	m_commandHandler				: i_commandHandler;					// Command handler function (via defined interface)
	
	// FiFo Command Buffer											
	m_FiFo							: FB_MemRingBuffer;					// FIFO command buffer
	m_CommandBuffer					: ARRAY[1..M_COMMAND_BUFFER_SIZE] OF BYTE;
	
	// Finite State Machine
									
	m_CommandInterfaceFsmTable		: ARRAY [0..COMMAND_FSM_STATE_ARRAY_MAX, 0..COMMAND_FSM_EVENT_ARRAY_MAX, 0..COMMAND_FSM_ACTIONS_ARRAY_MAX] OF BYTE := [
	
	(* FsmState_ControlFault -------------------------------------------------------------------------- *)
	(*  Next State											Action		   		                     *)
	
		(* FsmEvent_ControlEnable *)
		Command_FsmState.FsmState_ControlFault,				Command_FsmAction.FsmAction_None,
                          
		(* FsmEvent_ControlDisable *)
		Command_FsmState.FsmState_ControlDisabled,			Command_FsmAction.FsmAction_DisableControl,
		
		(* FsmEvent_RunCommand *)
		Command_FsmState.FsmState_ControlFault,				Command_FsmAction.FsmAction_None,
	
		(* FsmEvent_CommandDone *)
		Command_FsmState.FsmState_ControlFault,				Command_FsmAction.FsmAction_None,

		(* FsmEvent_Fault *)  
		Command_FsmState.FsmState_ControlFault,				Command_FsmAction.FsmAction_None,
		
		(* FsmEvent_Reset *)  
		Command_FsmState.FsmState_ControlDisabled,			Command_FsmAction.FsmAction_Reset
	,
	
	(* FsmState_ControlDisabled ----------------------------------------------------------------------- *)
	(*  Next State											Action		    		                    *)
	
		(* FsmEvent_ControlEnable *)
		Command_FsmState.FsmState_ControlReady,				Command_FsmAction.FsmAction_EnableControl,
                          
		(* FsmEvent_ControlDisable *)
		Command_FsmState.FsmState_ControlDisabled,			Command_FsmAction.FsmAction_None,
		
		(* FsmEvent_RunCommand *)
		Command_FsmState.FsmState_ControlDisabled,			Command_FsmAction.FsmAction_None,
	
		(* FsmEvent_CommandDone *)
		Command_FsmState.FsmState_ControlFault,				Command_FsmAction.FsmAction_None,

		(* FsmEvent_Fault *)  
		Command_FsmState.FsmState_ControlFault,				Command_FsmAction.FsmAction_Fault,
		
		(* FsmEvent_Reset *)  
		Command_FsmState.FsmState_ControlDisabled,			Command_FsmAction.FsmAction_Reset
  	,

	(* FsmState_CommandRunning ------------------------------------------------------------------------ *)
	(*  Next State											Action				                        *)
	
		(* FsmEvent_ControlEnable *)
		Command_FsmState.FsmState_CommandRunning,			Command_FsmAction.FsmAction_None,
                          
		(* FsmEvent_ControlDisable *)
		Command_FsmState.FsmState_ControlDisabled,			Command_FsmAction.FsmAction_DisableControl,
		
		(* FsmEvent_RunCommand *)
		FSM_EVENT_INVALID,									Command_FsmAction.FsmAction_Fault,
	
		(* FsmEvent_CommandDone *)
		FSM_STATE_CONDITIONAL,								Command_FsmAction.FsmAction_CommandDone,

		(* FsmEvent_Fault *)  
		Command_FsmState.FsmState_ControlFault,				Command_FsmAction.FsmAction_Fault,
		
		(* FsmEvent_Reset *)  
		Command_FsmState.FsmState_ControlDisabled,			Command_FsmAction.FsmAction_Reset
  	,

	(* FsmState_ControlReady -------------------------------------------------------------------------- *)
	(*  Next State											Action		                    		    *)
	
		(* FsmEvent_ControlEnable *)
		Command_FsmState.FsmState_ControlReady,				Command_FsmAction.FsmAction_None,
                          
		(* FsmEvent_ControlDisable *)
		Command_FsmState.FsmState_ControlDisabled,			Command_FsmAction.FsmAction_DisableControl,
		
		(* FsmEvent_RunCommand *)
		Command_FsmState.FsmState_CommandRunning,			Command_FsmAction.FsmAction_RunCommand,
	
		(* FsmEvent_CommandDone *)
		FSM_EVENT_INVALID,									Command_FsmAction.FsmAction_Fault,

		(* FsmEvent_Fault *)  
		Command_FsmState.FsmState_ControlFault,				Command_FsmAction.FsmAction_Fault,
		
		(* FsmEvent_Reset *)  
		Command_FsmState.FsmState_ControlDisabled,			Command_FsmAction.FsmAction_Reset
		
	];
	
	m_CommandInterfacelFSM			: fb_FSM(		fsmId			:= ADR(m_CommandInterfacelFSM),
													stateTable		:= ADR(m_CommandInterfaceFsmTable),
													actionHandler	:= THIS^, 	// Use a self pointer in order to keep the action handler routine (ExecuteAction) in same function block <JAISON>
													numStates		:= Command_FsmState.NUM_FsmCommandInterfaceStates,
													numEvents		:= Command_FsmEvent.NUM_FsmCommandInterfaceEvents,
													initialState	:= Command_FsmState.FsmState_ControlDisabled);
											
	m_CommandFsmError				: BOOL;								// FSM error bit (TRUE = FSM Halted)
	m_CommandFsmErrorNum			: TFsmError;						// FSM error ENUM number
	m_CommandFsmCurrentState		: Command_FsmState;					// Current FSM state output
	m_CommandFsmLastState			: Command_FsmState;					// Previous state used for debugging FSM errors
	m_CommandFsmLastEvent			: Command_FsmEvent;					// Last triggered event output
	m_CommandFsmLastAction			: Command_FsmAction;				// Last run action output
	
	m_CommandFsmTraceTable			: ARRAY[1..20] OF Command_FsmDebugTableEntry;
	
END_VAR
VAR CONSTANT
	(* DEFAULT COMMAND DEFINITIONS *)
	
	(* ----------------------------------------------------------------------------
	Const name  : M_COMMAND_NONE
	Description : Defined constant value for no command running.		
	Notes       : 
	---------------------------------------------------------------------------- *)
	M_COMMAND_NONE			: INT := 0;

	(* ----------------------------------------------------------------------------
	Const name  : M_COMMAND_RESET
	Description : Defined constant value for reset command.				
	Notes       : 
	---------------------------------------------------------------------------- *)
	M_COMMAND_RESET			: INT := -1;	
	
	(* ----------------------------------------------------------------------------
	Const name  : M_COMMAND_FAULT
	Description : Defined constant value for fault command.				
	Notes       : 
	---------------------------------------------------------------------------- *)
	M_COMMAND_FAULT			: INT := -2;	

		(* ----------------------------------------------------------------------------
	Const name  : M_RESPONSE_READY
	Description : Defined constant value for ready response.		
	Notes       : 
	---------------------------------------------------------------------------- *)
	M_RESPONSE_READY		: INT := 0;

	(* ----------------------------------------------------------------------------
	Const name  : M_RESPONSE_BUSY
	Description : Defined constant value for busy response.				
	Notes       : 
	---------------------------------------------------------------------------- *)
	M_RESPONSE_BUSY			: INT := -1;	
	
	(* ----------------------------------------------------------------------------
	Const name  : M_RESPONSE_FAULT
	Description : Defined constant value for fault response.				
	Notes       : 
	---------------------------------------------------------------------------- *)
	M_RESPONSE_FAULT		: INT := -2;	
	
	
	(* FIFO COMMAND BUFFER *)
	
	(* ----------------------------------------------------------------------------
	Const name  : M_COMMAND_BUFFER_NUM_ENTRIES
	Description : Maximum number of entries allocated for the FIFO buffer.			
	Notes       : Used in FIFO buffer size definition
	---------------------------------------------------------------------------- *)
	M_COMMAND_BUFFER_NUM_ENTRIES	: UINT := 20;
		
	(* ----------------------------------------------------------------------------
	Const name  : M_COMMAND_BUFFER_SIZE
	Description : Size in BYTES allocated for the FIFO buffer.			
	Notes       : Used in FIFO buffer initialization, Beckhoff adds 4 BYTES
				  to each entry into the buffer because each data set is complemented 
				  with additional information, so that it can be located later.
	---------------------------------------------------------------------------- *)
	M_COMMAND_BUFFER_SIZE	: UINT := M_COMMAND_BUFFER_NUM_ENTRIES * (SIZEOF(TControlCommandBuffer) + 4);
	
	(* Finite State Machine *)

	(* ----------------------------------------------------------------------------
	Const name  : FSM_NUM_EVENT_ACTIONS
	Description : Maximum number of actions that are to be executed for each event 
				  Must be at least 1 action defined				
	Notes       : Used in FSM table definitions
	---------------------------------------------------------------------------- *)
	COMMAND_FSM_NUM_EVENT_ACTIONS	: INT := 1;
	
	(* ----------------------------------------------------------------------------
	Const name  : FSM_NUM_STATES
	Description : Total number of states 
	Notes       : Used in FSM table definitions
	---------------------------------------------------------------------------- *)
	COMMAND_FSM_NUM_STATES			: INT := Command_FsmState.NUM_FsmCommandInterfaceStates;
	
	(* ----------------------------------------------------------------------------
	Const name  : FSM_NUM_EVENTS
	Description : Total number of events per state
	Notes       : Used in FSM table definitions
	---------------------------------------------------------------------------- *)
	COMMAND_FSM_NUM_EVENTS			: INT := Command_FsmEvent.NUM_FsmCommandInterfaceEvents;
	
	(* ----------------------------------------------------------------------------
	Const name  : FSM_STATE_ARRAY_MAX
	Description : Max state array index value in the FSM table
				  Must subtract 1 due to arrays starting at 0
	Notes       : Used in FSM table definitions
	---------------------------------------------------------------------------- *)
	COMMAND_FSM_STATE_ARRAY_MAX		: INT := COMMAND_FSM_NUM_STATES - 1;
	
	(* ----------------------------------------------------------------------------
	Const name  : FSM_EVENT_ARRAY_MAX
	Description : Max event array index value in the FSM table
				  Must subtract 1 due to arrays starting at 0
	Notes       : Used in FSM table definitions
	---------------------------------------------------------------------------- *)
	COMMAND_FSM_EVENT_ARRAY_MAX		: INT := COMMAND_FSM_NUM_EVENTS - 1;
	
	(* ----------------------------------------------------------------------------
	Const name  : FSM_ACTIONS_ARRAY_MAX
	Description : Max actions array index value in the FSM table
				  next state entry is element 0 
	Notes       : Used in FSM table definitions
	---------------------------------------------------------------------------- *)
	COMMAND_FSM_ACTIONS_ARRAY_MAX	: INT := COMMAND_FSM_NUM_EVENT_ACTIONS;
END_VAR

(* ---------------------------------------------------------------------------
Func name   : 	CMD_ClearCommandBuffer
Description : 	Resets the FIFO buffer and clears current command and
				all buffered commands.
Inputs      :	None
Returns     : 	TRUE
Notes       : 	Used when the command interface is reset.
--------------------------------------------------------------------------- *)

METHOD CMD_ClearCommandBuffer : BOOL
VAR_INPUT
END_VAR
// Clear the command buffer			
MEMSET			(	destAddr:= ADR(m_CommandBuffer) , 
				 	fillByte:= 0 , 
				 	n:= SIZEOF(m_CommandBuffer));	

// Clear the current command variable		
MEMSET			(	destAddr:= ADR(m_CurrentCommand) , 
				 	fillByte:= 0 , 
					n:=  SIZEOF(m_CurrentCommand));	

// Reset the command buffer					
m_FiFo.A_Reset();

CMD_ClearCommandBuffer := TRUE;
END_METHOD

(* ---------------------------------------------------------------------------
Func name   : 	CMD_Fault
Description : 	Faults the FSM and transitions to the "Fault" state.
				Commands will NO LONGER be processed.
Inputs      :	None
Returns     : 	None
Notes       : 	Can be used in the interface routines if an error
				occurs that warrants command processing to stop.
--------------------------------------------------------------------------- *)

METHOD CMD_Fault
VAR_INPUT
END_VAR
// FAULT- Send Fault event to FSM
m_CommandInterfacelFSM.FSM_ProcessEvent(event:= Command_FsmEvent.FsmEvent_Fault);
END_METHOD

(* ---------------------------------------------------------------------------
Func name   : 	CMD_Init
Description : 	Initialization routine to setup the command interface
Inputs      :	commandHandler	:	command handler functions pointer (via defined interface)
Returns     : 	None
Notes       : 	Should be run ONCE for each instantiation of the
				command interface. Usually in the FB_INIT method.
--------------------------------------------------------------------------- *)

METHOD CMD_Init
VAR_INPUT
	commandHandler		: i_commandHandler;		// Command handler function (via defined interface)
END_VAR
// Set the FSM error state
m_CommandInterfacelFSM.FSM_SetErrorState(Command_FsmState.FsmState_ControlFault);

// Clear all event triggers to ensure all events are captured on startup
m_EnableTrigger(CLK:= FALSE);
m_DisableTrigger(CLK:= FALSE);
m_CommandDoneTrigger(CLK:= FALSE);

// Clear all flags
xBusy 	:= FALSE;
xDone 	:= FALSE;
xFault	:= FALSE;

// Set initial Variables
m_ControlEnabled := FALSE;

// Initialize the Command Handler Function
m_commandHandler := commandHandler;

// FIFO initialization - Not Needed <REMOVE>
//m_FiFo.Initialize(pBuffer := ADR(m_CommandBuffer[1]), udiBufferSize := M_COMMAND_BUFFER_SIZE * SIZEOF(TControlCommandBuffer));
//m_FiFo(pBuffer := ADR(m_CommandBuffer[1]), cbBuffer := M_COMMAND_BUFFER_SIZE * SIZEOF(TControlCommandBuffer)); // TEST THIS

// Fsm Test Table
m_CommandInterfacelFSM.FSM_SetDebugTraceTable(	pDebugTable := ADR(m_CommandFsmTraceTable),
												uiTableSize := SIZEOF(m_CommandFsmTraceTable));
END_METHOD

(* ---------------------------------------------------------------------------
Func name   : 	CMD_IsCommandValid
Description : 	Determines the validity of a command input.
Inputs      :	command	:	command to check of type TControlCommand (INT)
Returns     : 	TRUE if command is valid, FALSE otherwise
Notes       : 	Valid commands are > 0
--------------------------------------------------------------------------- *)

METHOD CMD_IsCommandValid : BOOL
VAR_INPUT
	command		: TControlCommand;
END_VAR
// Check for valid command which is greater than 0.  
// NONE (0) and RESET (-1) are handled seperately. <JAISON>
IF command > 0 THEN
			
	CMD_IsCommandValid := TRUE;
				
ELSE
		
	// COMMAND INVALID
	CMD_IsCommandValid := FALSE;
		
END_IF
END_METHOD

(* ---------------------------------------------------------------------------
Func name   : 	CMD_Reset
Description : 	Sends reset command to the FSM and clears the trace table
				if configured.
Inputs      :	None
Returns     : 	None
Notes       : 	
--------------------------------------------------------------------------- *)

METHOD CMD_Reset
VAR_INPUT
END_VAR
// Send the Reset Command event to FSM
m_CommandInterfacelFSM.FSM_ProcessEvent(event:= Command_FsmEvent.FsmEvent_Reset);

// Clear the trace table
IF (m_pCmdTraceTable <> _NULL) THEN					
	MEMSET			(	destAddr	:= ADR(m_pCmdTraceTable) , 
						fillByte	:= 0 , 
				 		n			:=  SIZEOF(m_CmdTraceTableSize));	
END_IF
END_METHOD

(* ---------------------------------------------------------------------------
Func name   : 	CMD_SendCommand
Description : 	Sends the input command with Parms to the FIFO buffer
				to be processed by the interface.
Inputs      :	command	:	command ENUM type TControlCommand (INT)
				parms	:	pointer to command PARMS of type TControlCommandParms (ARRAY[1..12] OF WORD)
Returns     : 	TRUE on success, FALSE otherwise
Notes       : 	
--------------------------------------------------------------------------- *)

METHOD CMD_SendCommand : BOOL
VAR_INPUT
	command		: TControlCommand;
	parms		: POINTER TO TControlCommandParms;
END_VAR
VAR
	m_Command	: TControlCommandBuffer;
END_VAR
VAR CONSTANT
	nullParms	: TControlCommandParms := [0, 0, 0, 0, 0, 0, 0, 0, 0, 0, 0, 0];
END_VAR
// Handle special case of Reset Command - sends command directly to FSM
IF (command = M_COMMAND_RESET) THEN
	
	// Send the Reset Command event to FSM
	m_CommandInterfacelFSM.FSM_ProcessEvent(event:= Command_FsmEvent.FsmEvent_Reset);
	
	CMD_SendCommand := TRUE;

// Handle special case of None Command
ELSIF (command = M_COMMAND_NONE) THEN
	
	// DO NOTHING
	
	CMD_SendCommand := TRUE;
	
ELSIF (command = M_COMMAND_FAULT) THEN
	
	CMD_Fault();
	
	CMD_SendCommand := TRUE;

ELSIF (m_FiFo.nCount < M_COMMAND_BUFFER_NUM_ENTRIES) AND m_ControlEnabled AND CMD_IsCommandValid(command) THEN

	m_Command.command := command;
	
	IF (parms <> _NULL) THEN
		m_Command.parms := parms^;
	ELSE
		m_Command.parms := nullParms;
	END_IF
	
	// Clear Response Here
	MEMSET			(	destAddr	:= ADR(m_Command.response), 
						fillByte	:= 0, 
						n			:= SIZEOF(m_Command.response));
								
	m_FiFo.A_AddTail(pWrite := ADR(m_Command), cbWrite := SIZEOF(m_Command));
	
	CMD_SendCommand := TRUE;

ELSE
	
	CMD_SendCommand := FALSE;
	
END_IF
END_METHOD

(* ---------------------------------------------------------------------------
Func name   : 	CMD_SetTraceTable
Description : 	Sets the trace table for use with the CMD_TRACE function which
				tracks previously completed commands.
Inputs      :	pTraceTable			-	pointer to the trace table
				uiTableSize			-	size of the trace table array in BYTES
Returns     : 	TRUE on success, else FALSE
Notes       : 	When setting a trace table use the generic TControlCommandBuffer
				type in order to ensure the size is proper.  The derived class
				will be responsible for decoding the command/response INT values
				into more understandable ENUMs if required.
--------------------------------------------------------------------------- *)

METHOD CMD_SetTraceTable : BOOL
VAR_INPUT
	pTraceTable			: POINTER TO TControlCommandBuffer;		// Pointer to the trace table
	uiTableSize			: UINT;									// Size of the debug table array in BYTES
END_VAR
// Test to ensure the debug table size is dividible by BYTES so the pointer manipulation does not crash the system. <JAISON>
IF ((uiTableSize MOD SIZEOF(TControlCommandBuffer)) = 0) THEN
	
	// Clear the trace table				
	MEMSET		     (	destAddr	:= 	pTraceTable, 
				 		fillByte	:= 0 , 
						n			:=  uiTableSize);	

	// Set the trace table pointer
	m_pCmdTraceTable := pTraceTable;
	
	// Set the trace table size
	m_CmdTraceTableSize := uiTableSize;
	
	// Return TRUE
	CMD_SetTraceTable := TRUE;
	
ELSE
	
	// Return FALSE
	CMD_SetTraceTable := FALSE;
	
END_IF
END_METHOD

(* ---------------------------------------------------------------------------
Func name   : 	CMD_TRACE
Description : 	This method allows the command interface to trace previously
				completed commands in an externally defined trace table.
Inputs      :	command	-	pointer to the command buffer to be added
Returns     : 	None
Notes       : 	Initially the trace table pointer will be NULL, you must 
				run the CMD_SetTraceTable to initialize the functionality.
--------------------------------------------------------------------------- *)
METHOD CMD_TRACE

VAR_INPUT
	command 			: POINTER TO TControlCommandBuffer;	// The command to be added to the trace table
END_VAR
VAR
	m_NumCommands		: UINT;								// Calculated number of commands in the trace table
	m_Command			: TControlCommandBuffer;			// Copy of the current command
	Offset				: UINT;								// Trace table pointer offset variable
	pCurrent 			: POINTER TO TControlCommandBuffer;	// Pointer to the current array element, used for array shifting
	pPrevious			: POINTER TO TControlCommandBuffer;	// Pointer to the previous array element, used for array shifting
END_VAR
// Ensure the trace table has been initialized
IF ((m_pCmdTraceTable <> _NULL) AND (command <> _NULL)) THEN
	
	// Determine the number of commands in the debug table array
	m_NumCommands := m_CmdTraceTableSize / SIZEOF(TControlCommandBuffer);
	
	// Set the offset to point to the last element of the debug table array
	Offset := (m_NumCommands - 1) * SIZEOF(TControlCommandBuffer);
	
	// Shift all the previous states down by one element
	WHILE (Offset >  0) DO
		
		// Set the current and previous state pointers
		pCurrent := m_pCmdTraceTable + Offset;
		pPrevious := pCurrent - SIZEOF(TControlCommandBuffer);
		
		// Update the current state value to the previous value
		pCurrent^ := pPrevious^;
	
		// Move the offset up by one element
		Offset := Offset - SIZEOF(TControlCommandBuffer);
		
	END_WHILE
	
	// Copy command data to local variable					
	MEMCPY		( destAddr := ADR(m_Command),
				  srcAddr  := command,
				  n		   := SIZEOF(m_Command));	
				  
	// Set the current state as the first element in the debug trace table array
	m_pCmdTraceTable^ := m_Command;
	
END_IF
END_METHOD

(* ---------------------------------------------------------------------------
Func name   : 	CMD_UpdateCommandInterface
Description : 	Interface update routine which is required to be called
				on EACH PLC SCAN by the inherited class.  This method is
				responsible for updating the FIFO buffer and FSM.
Inputs      :	None
Returns     : 	None
Notes       : 	
--------------------------------------------------------------------------- *)

METHOD CMD_UpdateCommandInterface
VAR_INPUT
END_VAR
//Run the Module Finite State Machine Logic Block <JAISON>
m_CommandInterfacelFSM(xEnable:= xEnable, xError=> m_CommandFsmError, errorNum=> m_CommandFsmErrorNum);

//Set the current FSM State variable for testing the FSM state transitions <JAISON>
m_CommandFsmCurrentState := m_CommandInterfacelFSM.FSM_GetCurrentState();

m_CommandFsmLastState := m_CommandInterfacelFSM.FSM_GetPreviousState();

// Run the Module FiFo Buffer Logic Block <JAISON>
m_FiFo(	pBuffer		:= ADR(m_CommandBuffer), 
		cbBuffer	:= M_COMMAND_BUFFER_SIZE);

// Handle the FIFO command buffer ONLY when in the ModuleReady state
IF (m_FiFo.nCount > 0) AND (m_CommandFsmCurrentState = Command_FsmState.FsmState_ControlReady) THEN
	
	// Remove an element from the command buffer <JAISON>
	m_FiFo.A_RemoveHead(pRead:= ADR(m_CurrentCommand), cbRead:= SIZEOF(m_CurrentCommand));
	
	// Ensure command is valid
	// This step is superfluous as commands going into the buffer are screened,
	// however, this should catch any data issues with the buffer. <JAISON>
	IF CMD_IsCommandValid(m_CurrentCommand.command) THEN
		
		// Send the Run Command event to FSM - Parm is pointer to the current command
		m_CommandInterfacelFSM.FSM_ProcessEventWithParms(	event		:= Command_FsmEvent.FsmEvent_RunCommand, 
															parms		:= ADR(m_CurrentCommand), 
															parmSize	:= SIZEOF(ADR(m_CurrentCommand)));
	
	ELSE
		
		// Send Fault event to FSM
		m_CommandInterfacelFSM.FSM_ProcessEvent(event:= Command_FsmEvent.FsmEvent_Fault);
		
	END_IF
	
END_IF

// (* EVENT TRIGGERS *)

// Module enable trigger, basic FSM Event with no user parameters <JAISON>
m_EnableTrigger(CLK:= xEnable);
IF (m_EnableTrigger.Q)THEN
	m_CommandInterfacelFSM.FSM_ProcessEvent(event:= Command_FsmEvent.FsmEvent_ControlEnable);
END_IF

// Module disable trigger, basic FSM Event with no user parameters <JAISON>
m_DisableTrigger(CLK:= xEnable);
IF (m_DisableTrigger.Q)THEN
	m_CommandInterfacelFSM.FSM_ProcessEvent(event:= Command_FsmEvent.FsmEvent_ControlDisable);
END_IF

// Handle command continuous logic HERE
IF (xBusy) THEN
	m_CommandDoneTrigger(CLK:= m_commandHandler.CommandRunning(pCurrentCommand:= ADR(m_CurrentCommand)));
ELSE
	m_CommandDoneTrigger(CLK:= FALSE);
END_IF

// Command done trigger, basic FSM Event with no user parameters <JAISON>
IF (m_CommandDoneTrigger.Q)THEN
	m_CommandInterfacelFSM.FSM_ProcessEventWithParms(	event		:= Command_FsmEvent.FsmEvent_CommandDone, 
														parms		:= ADR(m_CurrentCommand), 
														parmSize	:= SIZEOF(ADR(m_CurrentCommand)));
END_IF
END_METHOD

(* ---------------------------------------------------------------------------
Func name   : 	ExecuteAction
Description : 	This method is a standardized handler for
				each action generated by the FSM
Inputs      :	p_FSM			-	pointer to the instantiation of the FSM object
				currentAction	-	current FSM action being processed
				currentEvent	-	current FSM event being processed
Returns     : 	BOOL			- 	result of action function
Notes       : 	The approach of using an interface enables the user 
				of the FSM to define and handle actions based 
				on their design and implementation.
				
				Return TRUE to change state, FALSE to remain in 
				the same state, unless the FSM has the alwaysChangeState
				set to TRUE, then it will change state regardless 
				of action handler return.
				
				If a conditional state is to be used this action handler
				routuine is responsible for setting the conditionalState 
				value using the FSM_SetConditionalState() function.
--------------------------------------------------------------------------- *)

METHOD ExecuteAction : BOOL
VAR_INPUT
	p_FSM			: POINTER TO fb_FSM;
	currentAction	: TFsmAction;
	currentEvent	: TFsmEventDesc;
END_VAR
VAR
	pCurrentCommand	: POINTER TO TControlCommandBuffer;		// Pointer to current command parms
	faultCommand	: TControlCommandBuffer;				// Fault command buffer
	resetCommand	: TControlCommandBuffer;				// Reset command buffer
END_VAR
CASE currentAction OF
		
	Command_FsmAction.FsmAction_None:
			
		// DO ACTION NONE
			
		// RETURN TRUE
		ExecuteAction := TRUE;
			
	Command_FsmAction.FsmAction_EnableControl:
		
		// DO ACTION ENABLE CONTROL
				
		CMD_ClearCommandBuffer();
		xDone 	:= FALSE;
		xBusy	:= FALSE;
		xFault	:= FALSE;
			
		// Enable the control
		m_ControlEnabled := TRUE;
			
		// RETURN TRUE
		ExecuteAction := TRUE;
		
	Command_FsmAction.FsmAction_DisableControl:
		
		// DO ACTION DISABLE CONTROL
			
		CMD_ClearCommandBuffer();
		xDone := FALSE;
		xBusy := FALSE;
			
		// Disable the control
		m_ControlEnabled := FALSE;
			
		// RETURN TRUE
		ExecuteAction := TRUE;
			
	Command_FsmAction.FsmAction_RunCommand:
		
		// DO ACTION RUN COMMAND
			
		// Event Parms are pointer to TControlCommandBuffer
		pCurrentCommand := currentEvent.parms;
			
		// Clear the last run command response
		MEMSET(				destAddr	:= ADR(pCurrentCommand^.response), 
							fillByte	:= 0 , 
							n			:=  SIZEOF(pCurrentCommand^.response));	
				
		// Set the response to show command is running
		pCurrentCommand^.response.response 	:= M_RESPONSE_BUSY;
		pCurrentCommand^.response.message 	:= TO_STRING("Command Running");
		
		// Handle command start logic HERE 
		IF (NOT m_commandHandler.CommandStart(pCurrentCommand:= pCurrentCommand)) THEN
									
			// COMMAND START ERROR - Send Fault event to FSM
			m_CommandInterfacelFSM.FSM_ProcessEvent(event:= Command_FsmEvent.FsmEvent_Fault);
			
		END_IF
			
		// Set output flags
		xBusy := TRUE;
		xDone := FALSE;
			
		// Reset command done flag
		m_CommandDoneTrigger(CLK:= FALSE);
			
		// RETURN TRUE
		ExecuteAction := TRUE;
			
	Command_FsmAction.FsmAction_CommandDone:
		
		// DO ACTION COMMAND DONE - CONDITIONAL STATE
			
		// Event Parms are pointer to TControlCommandBuffer
		pCurrentCommand := currentEvent.parms;
		
		// Handle command done logic HERE - Set the response - Set the next state
		IF (m_commandHandler.CommandDone(pCurrentCommand:= pCurrentCommand)) THEN
				
			p_FSM^.FSM_SetConditionalState(state:= Command_FsmState.FsmState_ControlReady);
			
		ELSE
			
			// COMMAND DONE ERROR - Send Fault event to FSM
			m_CommandInterfacelFSM.FSM_ProcessEvent(event:= Command_FsmEvent.FsmEvent_Fault);
			
		END_IF
			
		// Set output flags
		xBusy := FALSE;
		xDone := TRUE;
			
		// Reset command done flag
		m_CommandDoneTrigger(CLK:= FALSE);
						
		// Add the current command/response to the trace table
		CMD_TRACE(command:= pCurrentCommand);
			
		// RETURN TRUE
		ExecuteAction := TRUE;
			
	Command_FsmAction.FsmAction_Fault:
		
		// DO ACTION FAULT
			
		// Disable the control
		m_ControlEnabled := FALSE;
		
		xFault	:= TRUE;
			
		// Modify the current response message to show fault
		m_CurrentCommand.response.response	:= M_RESPONSE_FAULT;
		m_CurrentCommand.response.message	:= TO_STRING("COMMAND INTERFACE FAULTED");
			
		// Copy the current command data, to show the command 
		// running when the fault occured; if any.		
		faultCommand.command 			:= m_CurrentCommand.command;
		faultCommand.parms				:= m_CurrentCommand.parms;
	
		// Modify the response to show that this is a fault event
		faultCommand.response.response 	:= M_RESPONSE_FAULT;
		faultCommand.response.message 	:= TO_STRING("COMMAND INTERFACE FAULTED");
			
		CMD_TRACE(command:= ADR(faultCommand));
			
		// Call Interface Fault function
		m_commandHandler.Fault();
			
		// RETURN TRUE
		ExecuteAction := TRUE;
		
	Command_FsmAction.FsmAction_Reset:
		
		// DO ACTION RESET
			
		CMD_ClearCommandBuffer();
			
		xDone 	:= FALSE;
		xBusy 	:= FALSE;
		xFault	:= FALSE;
			
		// Copy the current command data, to show the command 
		// is a reset command		
		resetCommand.command 			:= M_COMMAND_RESET;
	
		// Modify the response to show that the reset occured
		resetCommand.response.response 	:= M_RESPONSE_READY;
		resetCommand.response.message 	:= TO_STRING("COMMAND INTERFACE RESET");
			
		CMD_TRACE(command:= ADR(resetCommand));
		
		// Call Interface Reset function
		m_commandHandler.Reset();
			
		// Reset enable trigger to capture enable event
		m_EnableTrigger(CLK:= FALSE);
			
		// RETURN TRUE
		ExecuteAction := TRUE;	
				
	FSM_ACTION_UNEXPECTED_EVENT:
			
		// DO ACTION UNEXPECTED EVENT
		
		// ERROR TRAP - UNKNOWN ACTION
		// NOTE: 	This will HALT the FSM when it FAILS which is likely advisable here because
		//			this is a critical design time error.  All actions need to be defined, even
		//			if they simply log an event occured. <JAISON>
		p_FSM^.FSM_ASSERT(FALSE, TFsmError.FSM_INVALID_ACTION);
			
		// RETURN FALSE
		ExecuteAction := FALSE;
			
	FSM_ACTION_ERROR_EVENT:
		
		// DO ACTION ERROR EVENT
			
		// This action is executed when an FSM ASSERT Fails and the FSM is transitioning to the defined error state. <JAISON>
			
		// RETURN FALSE - This is irrelevant because the FSM will automatically transition to the error state.
		ExecuteAction := FALSE;
				
ELSE
			
	// ERROR TRAP - UNKNOWN ACTION
	// NOTE: 	This will HALT the FSM when it FAILS which is likely advisable here because
	//			this is a critical design time error.  All actions need to be defined, even
	//			if they simply log an event occured. <JAISON>
	p_FSM^.FSM_ASSERT(FALSE, TFsmError.FSM_INVALID_ACTION);
			
	// RETURN FALSE
	ExecuteAction := FALSE;
			
END_CASE;
	
m_CommandFsmLastEvent := currentEvent.event;
m_CommandFsmLastAction := currentAction;
m_CommandFsmLastState := p_FSM^.FSM_GetPreviousState();
END_METHOD

END_FUNCTION_BLOCK

// 20 Program Organization Units/FSM/Interfaces/i_actionHandler
(*AUTHOR:			Jaison Schaab*)
(*DATE:				December. 30 / 2019*)
(*DESCRIPTION: 		This is a standardized interface used by the FSM function
					block to handle generated actions*)
					
(*NOTES:      	 	All methods definied by this interface are required to
					be implimented by the user defined action handler
					function block.  Each methods inputs/outputs need
					to match exactly what is defined by the interface.
					
					The FSM requires the user defined function block which
					impliments this interface  to be passed into its 
					constructor upon instantiation.*)

INTERFACE i_actionHandler

(* ---------------------------------------------------------------------------
Func name   : 	ExecuteAction
Description : 	This method is a standardized handler for
				each action generated by the FSM
Inputs      :	p_FSM			-	pointer to the instantiation of the FSM object
				currentAction	-	current FSM action being processed
				currentEvent	-	current FSM event being processed
Returns     : 	BOOL			- 	result of action function
Notes       : 	The approach of using an interface enables the user 
				of the FSM to define and handle actions based 
				on their design and implementation.
				
				Return TRUE to change state, FALSE to remain in 
				the same state, unless the FSM has the alwaysChangeState
				set to TRUE, then it will change state regardless 
				of action handler return.
				
				If a conditional state is to be used this action handler
				routuine is responsible for setting the conditionalState 
				value using the FSM_SetConditionalState() function.
--------------------------------------------------------------------------- *)

METHOD ExecuteAction : BOOL
VAR_INPUT
	p_FSM			: POINTER TO fb_FSM;
	currentAction	: TFsmAction;
	currentEvent	: TFsmEventDesc;
END_VAR
END_METHOD

END_INTERFACE

// 20 Program Organization Units/FSM/fb_FSM
(*AUTHOR:			Jaison Schaab*)
(*DATE:				December 30 / 2019*)
(*DESCRIPTION: 		This Function Block provides a standard base functionality for
					a generic table driven finite state machine (FSM)*)
					
(*NOTES:			The user of the FSM function block is required to define the following:
					STATE ENUM of TYPE FsmState (BYTE) 		- 	List of desired states starting at 0 with the last entry being "NUM_FsmTestStates"
					EVENT ENUM of TYPE FsmEvent (BYTE) 		- 	List of desired events starting at 0 with the last entry being "NUM_FsmTestEvents"
					ACTION ENUM of TYPE FsmAction (BYTE) 	- 	List of desired actions starting at 0 with the last entry being "NUM_FsmTestActions"
					
					****The IEC Standard does NOT allow the ENUMERATION types to be defined as a non-registered type (ex. FsmState)
						To work around this simply define the required ENUMERATIONS as BYTE and remove the 
						"{attribute 'strict'}" from the header so that the system will correlate the non-registered types****
					
					Action Handler function block  			- 	user defined function block which impliments the i_actionHandler interface and
																will perform all required actions that are associated with events.
																
					****EVENTS may have parameters associated with them, ACTIONS DO NOT.  The user is required to define their own
						parameter types which can be associated with events and passed into the action handler.****									
					
					****TO TRIGGER EVENTS use the FSM methods "FSM_ProcessEvent" OR "FSM_ProcessEventWithParms"****
					****Calling the "FSM_Reset" method will RESET the FSM back to the default constructor state
						This is required after any FSM error as the FSM block will cease to function until a RESET occurs****
*)

(*UPDATE: 			March. 18 2021 - Jaison Schaab

					Code Ported from Wago.
					
					Code has NOT Yet been tested.
*)

FUNCTION_BLOCK fb_FSM
VAR_INPUT
	xEnable				: BOOL;											// Function block enable - TRUE to enable FSM functionality
END_VAR
VAR_OUTPUT
	xError				: BOOL;											// FSM error state output, if TRUE FSM will cease operation until reset (FSM_ASSERT sets state)
	errorNum			: TFsmError;									// The enumeration value describing the failed assert (type FsmError) 
END_VAR
VAR
	(* Fsm Desc *)
	m_fsmId				: POINTER TO fb_FSM;							// Pointer to the instantiation of the FSM object
	
	m_currentState		: TFsmState;									// Current state id of the FSM
	m_prevState			: TFsmState;									// Memory of the previously ran state used for debugging errors
	m_initialState		: TFsmState;									// Internal memory of the initial state id, used for FSM reset
	m_errorState		: TFsmState;									// Internal memory of an error state id, used when FSM Assert fails
	
	m_conditionalState	: TFsmState;									// Conditional next state parameter - set by action handler
	m_alwaysChangeState	: BOOL;											// Internal state change flag for conditional states - when TRUE action handler return is ignored
	
	m_numStates			: UINT;											// Number of states in the FSM
	m_numEvents			: UINT;											// Number of events defined for the FSM
	
	m_stateTable		: POINTER TO TFsmState;							// Pointer to the FSM table
	m_eventEntrySize	: UINT;											// Size of an event entry in the FSM table, consists of one event type and one action type
	m_stateEntrySize	: UINT;											// Size of a state entry in the FSM table, consists of numEvents * event entry size
	
	m_eventQ			: ARRAY[0.._FSM_EVENT_Q_SIZE] OF TFsmEventDesc;	// Event queue array, utilized as a circular buffer
	m_eventQPutIndex	: TFsmEventQIndex;								// Event queue index used for inserting events
	m_eventQGetIndex	: TFsmEventQIndex;								// Event queue index used for removing events
	m_numInEventQ		: TFsmEventQIndex;								// Current number of events in the queue
	
	m_FsmActionHandler	: i_actionHandler;								// Action handler function (via defined interface)
	
	(* Internal *)
	m_nextState 		: TFsmState;									// Internal variable used to track the next state transition
	m_changeState		: BOOL := TRUE;									// Internal state change flag used when processing events
	m_currentEvent		: TFsmEventDesc;								// Current FSM event being processed
	m_currentAction		: TFsmAction;									// Current FSM action id being processed
	
	m_pFsmDebugTable	: POINTER TO TFsmDebugTableEntry;				// Pointer to the debug table
	m_FsmDebugTableSize	: UINT;											// Size of the debug table array in BYTES
	m_StateChangeTimer	: fb_ElapsedTime;								// Timer to track the time between state changes in debug table
	
END_VAR

(* Handle the events *)
WHILE ((xEnable) AND (m_numInEventQ <> 0) AND (NOT xError)) DO
  
	m_changeState := TRUE;						// Assume we are going to change state
	m_conditionalState := FSM_STATE_INVALID; 	// Assume the conditional state is invalid to ensure the action function sets it
	
	m_currentEvent := FSM_GetCurrentEvent();
	m_currentAction := FSM_GetCurrentAction(state:= m_currentState, event:= m_currentEvent);
	
	m_prevState := m_CurrentState;				// Set the previous state for debugging FSM errors
	
	(* FSM TRACE HANDLE EVENT *)
	
	(* unexpected action, do not change state *)
	IF (m_currentAction = FSM_ACTION_UNEXPECTED_EVENT) THEN
		
		(* FSM TRACE UNEXPECTED ACTION *)
		m_changeState := FALSE;	
	
	END_IF
	
	(* FSM TRACE EXECUTE ACTION *)
	
	(* process the action, returning true means change state, but check the change state flag *)
	IF (NOT m_FsmActionHandler.ExecuteAction(p_FSM:= m_fsmId, currentAction:= m_currentAction, currentEvent:= m_currentEvent)) THEN
		
		// Action Handler Returned FALSE
		IF (_FSM_ALLOW_CONDITIONAL_STATES) THEN
			
			(* maybe change state on a FALSE return *)
			IF (m_alwaysChangeState =  FALSE) THEN
					
				m_changeState := FALSE;
				
			END_IF
				
		ELSE
			
		// Never change state on a FALSE return
        m_changeState := FALSE;
			
		END_IF
		
	END_IF (* end - (actions) *)
	
	(* Change state *)
	IF (m_changeState) THEN
    
		m_nextState := FSM_GetNextState(state:= m_currentState, event:= m_currentEvent);

		(* 	get the next state dynamically from the action handler 
			if allowed and conditional state entered into table. *)
		IF ((_FSM_ALLOW_CONDITIONAL_STATES) AND (m_nextState = FSM_STATE_CONDITIONAL)) THEN

			m_nextState := m_conditionalState;
		
		END_IF
      
		(* validate the next state value *)
		FSM_ASSERT(BYTE_TO_UINT(m_nextState) < m_numStates, TFsmError.FSM_INVALID_NEXT_STATE);
		
		// If next state is invalid, stay in same state - Assert above will set xError flag
		// Ignore this if the FSM_ASSERT already set the current state to the error state <JAISON>
		IF ((xError) AND (m_currentState <> m_errorState) )THEN
			(* stay in the same state *)
			m_nextState := m_currentState;
		END_IF
    
	ELSE
    
		(* stay in the same state *)
		m_nextState := m_currentState;
		
	END_IF
    
    
	(* move to the next state *)
	IF (m_nextState <> m_currentState) THEN
		
		m_currentState := m_nextState;
    
	END_IF
	
	// Trace the FSM Event
	FSM_TRACE(state:= m_currentState, event:= m_currentEvent);
	
	(* remove this message *)
	m_numInEventQ := m_numInEventQ - 1;

	(* get the next FSM message *)
	m_eventQGetIndex := m_eventQGetIndex + 1;
	IF (m_eventQGetIndex = _FSM_EVENT_Q_SIZE) THEN
    
		m_eventQGetIndex := 0;
		
	END_IF

END_WHILE	(* end of while *)

(* ---------------------------------------------------------------------------
Func name   : 	FB_exit
Description : 	Destructor
Inputs      :	None
Returns     : 	None
Notes       : 	
--------------------------------------------------------------------------- *)

METHOD FB_exit : BOOL
VAR_INPUT
	bInCopyCode : BOOL; // if TRUE, the exit method is called for exiting an instance that is copied afterwards (online change)
END_VAR
// Do nothing
END_METHOD

(* ---------------------------------------------------------------------------
Func name   : 	FB_init
Description : 	Constructor
Inputs      :	fsmId			-	pointer to the instatiation of the FSM object
				stateTable		-	pointer to the FSM table
				actionHandler	-	action handler function (via defined interface)
				numStates		-	number of states in the FSM
				numEvents		-	number of events defined for the FSM				
				initialState	-	initial state for the FSM
Returns     : 	None
Notes       : 	
--------------------------------------------------------------------------- *)

METHOD FB_init : BOOL
VAR_INPUT
	bInitRetains 		: BOOL; 				// if TRUE, the retain variables are initialized (warm start / cold start)
    bInCopyCode  		: BOOL; 				// if TRUE, the instance afterwards gets moved into the copy code (online change)
	fsmId				: POINTER TO fb_FSM;	// Pointer to the instatiation of the FSM object
	stateTable			: POINTER TO TFsmState; // Pointer to the FSM table
	actionHandler		: i_actionHandler;		// Action handler function (via defined interface)
	numStates			: UINT;					// Number of states in the FSM
	numEvents			: UINT;					// Number of events defined for the FSM
	initialState		: TFsmState;			// Initial state for the FSM
END_VAR
// initialize a self pointer to allow the action handler to access FSM functions
m_fsmId := fsmId;

// Initialize the initial (START) state
m_initialState := initialState;
m_currentState := initialState;

m_errorState := FSM_STATE_INVALID; // Should this be a constructor value??
m_prevState	:= FSM_STATE_INVALID;
m_currentAction := FSM_ACTION_NONE;

// Initialize the conditional state to invalid - force the action handler to set it
m_conditionalState := FSM_STATE_INVALID;
m_alwaysChangeState := FALSE;

m_numStates := numStates;
m_numEvents := numEvents;

// Initialize the state table
m_stateTable := stateTable;
m_eventEntrySize := SIZEOF(TFsmState) + SIZEOF(TFsmAction);
m_stateEntrySize := m_numEvents * m_eventEntrySize;

// Initialize event queue
MEMSET(destAddr:= ADR(m_eventQ), fillByte:= 0, n:= SIZEOF(m_eventQ));
m_eventQPutIndex := 0; 
m_eventQGetIndex := 0;
m_numInEventQ := 0;

// Initialize the current event to be the num events
m_currentEvent.event	:= TO_BYTE(m_numEvents);
m_currentEvent.parms	:= 0;
m_currentEvent.parmSize	:= 0;

// Initialize the Action Handler Function
m_FsmActionHandler := actionHandler; 

// Initialize error handling
xError := FALSE;
errorNum := TFsmError.FSM_ERROR_NONE;

// Initialize the debug trace table to NULL
m_pFsmDebugTable := 0;
m_FsmDebugTableSize	:= 0;
END_METHOD

(* ---------------------------------------------------------------------------
Func name   : 	FSM_ASSERT
Description : 	This method allows FSMs to handle assert conditions.
Inputs      :	condition	-	condition to assert
				error		-	enumerated error value of type FsmError
Returns     : 	BOOL		-	the input condition is reflected as the function return
								TRUE means the assert passed, FALSE means it failed
Notes       : 	When an assert fails the FSM will be halted until it is reset.
--------------------------------------------------------------------------- *)

METHOD FSM_ASSERT : BOOL
VAR_INPUT
	condition	: BOOL;
	error		: TFsmError;
END_VAR
IF (NOT condition) THEN
	
	// Set the error bit to TRUE which will halt state machine operation
	xError := TRUE;
	errorNum := error;
	
	// If an error state has been set transition the FSM to that state
	IF (m_errorState <> FSM_STATE_INVALID) THEN
	
		// process the FSM_ACTION_ERROR_EVENT action, ignore the return condition as the FSM will automatically transition to the error state. <JAISON>
		m_FsmActionHandler.ExecuteAction(p_FSM:= m_fsmId, currentAction:= FSM_ACTION_ERROR_EVENT, currentEvent:= m_currentEvent);
	
		// Set the current and next state
		m_currentState := m_nextState := m_errorState;
	
		// Trace the state transition
		FSM_TRACE(state:= m_currentState, event:= m_currentEvent);
	
	END_IF

END_IF

// Return condition value
FSM_ASSERT := condition;
END_METHOD

(* ---------------------------------------------------------------------------
Func name   : 	FSM_GetCurrentAction
Description : 	Retrieves the current action of the FSM.
Inputs      :	state		- 	current FSM state
				event		- 	current triggered event
Returns     : 	FsmAction	- 	the current FSM action associated with
								the input event/action
Notes       : 	
--------------------------------------------------------------------------- *)

METHOD PRIVATE FSM_GetCurrentAction : TFsmAction
VAR_INPUT
	state					: TFsmState;
	event					: TFsmEventDesc;
END_VAR
VAR
	m_state_offset			: UINT;
	m_event_offset			: UINT;
	p_CurrentAction			: POINTER TO TFsmAction;
END_VAR
VAR CONSTANT
	FSM_TABLE_ACTION_ENTRY 	: UINT := 1;
END_VAR
m_state_offset := state * m_stateEntrySize;
m_event_offset := event.event * m_eventEntrySize;

p_CurrentAction := m_stateTable + m_state_offset + m_event_offset + FSM_TABLE_ACTION_ENTRY;

FSM_GetCurrentAction := p_CurrentAction^;
END_METHOD

(* ---------------------------------------------------------------------------
Func name   : 	FSM_GetCurrentEvent
Description : 	Retrieves the current action of the FSM.
Inputs      :	None
Returns     : 	FsmEventDesc	- 	the current FSM event
Notes       : 	This function is intended to be called from 
             	an action routine
--------------------------------------------------------------------------- *)

METHOD FSM_GetCurrentEvent : TFsmEventDesc
VAR_INPUT
END_VAR
FSM_GetCurrentEvent := m_eventQ[m_eventQGetIndex];
END_METHOD

(* ---------------------------------------------------------------------------
Func name   : 	FSM_GetCurrentState
Description : 	Retrieves the current state of the FSM.
Inputs      :	None
Returns     : 	FsmState	-	the current FSM state or 
								FSM_STATE_INVALID on error 
Notes       : 	This function is intended to be called from 
              	an action routine
--------------------------------------------------------------------------- *)

METHOD FSM_GetCurrentState : TFsmState
VAR_INPUT
END_VAR
FSM_GetCurrentState := m_currentState;
END_METHOD

(* ---------------------------------------------------------------------------
Func name   : 	FSM_GetNextState
Description : 	Retrieves the next state from the FSM.
Inputs      :	state		- 	current FSM state
				event		- 	current triggered event
Returns     : 	FsmState	- 	the current FSM next state associated with
								the input event/action
Notes       : 	
--------------------------------------------------------------------------- *)

METHOD PRIVATE FSM_GetNextState : TFsmState
VAR_INPUT
	state						: TFsmState;
	event						: TFsmEventDesc;
END_VAR
VAR
	m_state_offset				: UINT;
	m_event_offset				: UINT;
	p_NextState					: POINTER TO TFsmState;
END_VAR
VAR CONSTANT
	FSM_TABLE_NEXT_STATE_ENTRY 	: UINT := 0;
END_VAR
m_state_offset := state * m_stateEntrySize;
m_event_offset := event.event * m_eventEntrySize;

p_NextState := m_stateTable + m_state_offset + m_event_offset + FSM_TABLE_NEXT_STATE_ENTRY;

FSM_GetNextState := p_NextState^;
END_METHOD

(* ---------------------------------------------------------------------------
Func name   : 	FSM_GetPreviousState
Description : 	Retrieves the previous state of the FSM.
Inputs      :	None
Returns     : 	FsmState	-	the previous FSM state or 
								FSM_STATE_INVALID on error 
Notes       : 	This function is intended to be called from 
              	an action routine
--------------------------------------------------------------------------- *)

METHOD FSM_GetPreviousState : TFsmState
VAR_INPUT
END_VAR
FSM_GetPreviousState := m_prevState;
END_METHOD

(* ---------------------------------------------------------------------------
Func name   :	FSM_ProcessEvent
Description : 	Sends an event to the FSM.
Inputs      : 	event	-	the FSM event Id
Returns     :	TRUE on success, else FALSE
Notes       : 	There are no parameters associated with these events
--------------------------------------------------------------------------- *)

METHOD FSM_ProcessEvent : BOOL
VAR_INPUT 
	event		: TFsmEvent;
END_VAR
IF (xEnable) THEN
	
	// Simply call the Process Event with Parms using a NULL pointer for the parms
	FSM_ProcessEventWithParms(event:= event, parms:= 0, parmSize:= 0);
	
	FSM_ProcessEvent := TRUE;
	
ELSE
	
	FSM_ProcessEvent := FALSE;
	
END_IF
END_METHOD

(* ---------------------------------------------------------------------------
Func name   : FSM_ProcessEventWithParms
Description : Sends an event, with parameters, to the FSM.
Inputs      : event		-	the FSM event id
              parms		-	byte pointer to the parameter structure for the event
              parmSize	-	the size of the parameter structure in bytes
Returns     : TRUE on success, else FALSE
Notes       : This function assume that the producer and consumer of
              the message Queue are mutually exclusive
--------------------------------------------------------------------------- *)

METHOD FSM_ProcessEventWithParms : BOOL
VAR_INPUT
	event			: TFsmEvent;
	parms			: POINTER TO BYTE;
	parmSize		: UINT;
END_VAR
VAR

END_VAR
(* validate the size of the parameter struct *)
FSM_ASSERT(parmSize <= _FSM_MAX_PARM_STRUCT_SIZE, TFsmError.FSM_PARM_SIZE_ERROR);
	
(* validate the maximum event Q size is not exceeded *)
FSM_ASSERT(m_numInEventQ < TO_UINT(_FSM_EVENT_Q_SIZE), TFsmError.FSM_EVENT_Q_SIZE_ERROR);
	
(* validate the event being processed value *)
FSM_ASSERT(event <= m_numEvents, TFsmError.FSM_INVALID_EVENT_ERROR);

IF ((xEnable) AND (NOT xError)) THEN
	
	(* Store the new event in the eventQ *)
	m_eventQ[m_eventQPutIndex].event := event;
	m_eventQ[m_eventQPutIndex].parms := parms;
	m_eventQ[m_eventQPutIndex].parmSize := parmSize;
	
	(*FSM TRACE Q EVENT*)
	
	(* Update the put pointer *)
	m_eventQPutIndex := m_eventQPutIndex + 1;
	IF (m_eventQPutIndex = TO_UINT(_FSM_EVENT_Q_SIZE)) THEN
		m_eventQPutIndex := 0;
	END_IF
	
	m_numInEventQ := m_numInEventQ + 1;
	
	FSM_ProcessEventWithParms := TRUE;

ELSE
	
	(* block NOT enabled or error flag set *)
	FSM_ProcessEventWithParms := FALSE;
	
END_IF
END_METHOD

(* ---------------------------------------------------------------------------
Func name   : 	FSM_Reset
Description : 	Routine to reset the FSM back to its initial (START) state.
Inputs      :	None
Returns     : 	None
Notes       : 	This will reset all event Q data as well
--------------------------------------------------------------------------- *)

METHOD FSM_Reset
VAR_INPUT
END_VAR
// Initialize the initial (START) state
m_currentState := m_initialState;
m_currentAction := FSM_ACTION_NONE;

m_prevState	:= FSM_STATE_INVALID;

// Trace the state transition
FSM_TRACE(state:= m_currentState, event:= m_currentEvent);

// Initialize the conditional state to invalid - force the action handler to set it
m_conditionalState := FSM_STATE_INVALID;

(* Initialize Event Queue *)
MEMSET(destAddr:= ADR(m_eventQ), fillByte:= 0, n:= SIZEOF(m_eventQ));
m_eventQPutIndex := 0; 
m_eventQGetIndex := 0;
m_numInEventQ := 0;

// Initialize the current event to be the num events
m_currentEvent.event	:= TO_BYTE(m_numEvents);
m_currentEvent.parms	:= 0;
m_currentEvent.parmSize	:= 0;

(* Initialize Error Handling *)
xError := FALSE;
errorNum := TFsmError.FSM_ERROR_NONE;
END_METHOD

(* ---------------------------------------------------------------------------
Func name   : 	FSM_SetAlwaysChangeState
Description : 	Sets the state change flag for conditional states.
Inputs      :	enable - state of the flag
Returns     : 	TRUE on success, else FALSE
Notes       : 	Enabling this flag will allow conditional states to
              	always transition regardless of the action function
              	return value.
--------------------------------------------------------------------------- *)

METHOD FSM_SetAlwaysChangeState : BOOL
VAR_INPUT
	enable	: BOOL;
END_VAR
m_alwaysChangeState := enable;

FSM_SetAlwaysChangeState := TRUE;
END_METHOD

(* ---------------------------------------------------------------------------
Func name   : 	FSM_SetConditionalState
Description : 	Sets the condition state for the FSM.
Inputs      :	state	-	the state to transition to after event processing
Returns     : 	TRUE on success, else FALSE
Notes       : 	In conditional states, the state is set by the action
              	function. This interface allows the action function to
             	set the state. Not setting the state in a conditional
              	state will invoke an FSM assertion and error the FSM.  
--------------------------------------------------------------------------- *)

METHOD FSM_SetConditionalState : BOOL
VAR_INPUT
	state		: TFsmState;
END_VAR
(* validate the next state value *)
IF (FSM_ASSERT(BYTE_TO_UINT(state) < m_numStates, TFsmError.FSM_INVALID_CONDITIONAL_STATE)) THEN
	m_conditionalState := state;

	// Return TRUE
	FSM_SetConditionalState := TRUE;
	
ELSE
		
	// Return FALSE
	FSM_SetConditionalState := FALSE;
	
END_IF
END_METHOD

(* ---------------------------------------------------------------------------
Func name   : 	FSM_SetDebugTraceTable
Description : 	Sets the debug table for use with the FSM_TRACE function in FSM.
Inputs      :	pFsmDebugTable		-	pointer to the debug table
				uiFsmDebugTableSize	-	size of the debug table array in BYTES
Returns     : 	TRUE on success, else FALSE
Notes       : 	When setting a debug table use the specific state ENUM
				type instead of a simple BTYE array for more understandable
				state entries.
--------------------------------------------------------------------------- *)

METHOD FSM_SetDebugTraceTable : BOOL
VAR_INPUT
	pDebugTable			: POINTER TO TFsmState;		// Pointer to the debug table
	uiTableSize			: UINT;						// Size of the debug table array in BYTES
END_VAR
// Test to ensure the debug table size is dividible by BYTES so the pointer manipulation does not crash the system. <JAISON>
IF ((uiTableSize MOD SIZEOF(TFsmState)) = 0) THEN
	
	// Preset the Debug Table
	MEMSET(destAddr:= pDebugTable, fillByte:= 16#FF, n:= uiTableSize);

	// Set the debug table pointer
	m_pFsmDebugTable := pDebugTable;
	
	// Set the debug table size
	m_FsmDebugTableSize := uiTableSize;
	
	// Set the initial start time for the state change timer
	m_StateChangeTimer.StartNow();
	
	// Add the current state to the Debug Table as a starting point for debugging
	FSM_TRACE(state:= m_currentState, event:= m_currentEvent);
	
	// Return TRUE
	FSM_SetDebugTraceTable := TRUE;
	
ELSE
	
	// Return FALSE
	FSM_SetDebugTraceTable := FALSE;
	
END_IF
END_METHOD

(* ---------------------------------------------------------------------------
Func name   : 	FSM_SetErrorState
Description : 	Sets the error state of the FSM.
Inputs      :	state	-	the state to transition to after FSM Assert fails
Returns     : 	TRUE on success, else FALSE
Notes       : 	The error state is set to FSM_STATE_INVALID as default
				which will keep the FSM in its current state on error.
				However, if the user wants a particular error state to be
				entered in the event of an error they can use this method
				to set it.
--------------------------------------------------------------------------- *)

METHOD FSM_SetErrorState : BOOL
VAR_INPUT
	state		: TFsmState;
END_VAR
// validate the error state value
IF (FSM_ASSERT(BYTE_TO_UINT(state) < m_numStates, TFsmError.FSM_INVALID_ERROR_STATE)) THEN

	m_errorState := state;

	// Return TRUE
	FSM_SetErrorState := TRUE;
	
ELSE
		
	// Return FALSE
	FSM_SetErrorState := FALSE;
	
END_IF
END_METHOD

(* ---------------------------------------------------------------------------
Func name   : 	FSM_TRACE
Description : 	This method allows the FSM to trace state transitions in
				and externally defined debug trace table.
Inputs      :	state	-	the FSM state to be added to the debug trace table
				event	-	the FSM event to be added to the debug trace table
Returns     : 	None
Notes       : 	Initially the debug table will be NULL, you must run the
				FSM_SetDebugTraceTable to initialize the functionality.
				
				This method is called within the FSM whenever a state changes.
--------------------------------------------------------------------------- *)

METHOD FSM_TRACE
VAR_INPUT
	state 				: TFsmState;						// The FSM state to be added to the debug trace table
	event				: TFsmEventDesc;					// The FSM event to be added to the debug trace table
END_VAR
VAR
	m_NumTraceStates	: UINT;								// Calculated number of states in the debug trace table
	Offset				: UINT;								// Debug trace table pointer offset variable
	pCurrent 			: POINTER TO TFsmDebugTableEntry;	// Pointer to the current array element, used for array shifting
	pPrevious			: POINTER TO TFsmDebugTableEntry;	// Pointer to the previous array element, used for array shifting
END_VAR
// Ensure the debug table has been initialized
IF (m_pFsmDebugTable <> 0) THEN
	
	// Determine the number of states in the debug table array
	m_NumTraceStates := m_FsmDebugTableSize / SIZEOF(TFsmDebugTableEntry);
	
	// Set the offset to point to the last element of the debug table array
	Offset := (m_NumTraceStates - 1) * SIZEOF(TFsmDebugTableEntry);
	
	// Shift all the previous states down by one element
	WHILE (Offset >  0) DO
		
		// Set the current and previous state pointers
		pCurrent := m_pFsmDebugTable + Offset;
		pPrevious := pCurrent - SIZEOF(TFsmDebugTableEntry);
		
		// Update the current state value to the previous value
		pCurrent^ := pPrevious^;
	
		// Move the offset up by one element
		Offset := Offset - SIZEOF(TFsmDebugTableEntry);
		
	END_WHILE
	
	// Set the first element in the debug trace table array
	
	// Set the state
	m_pFsmDebugTable^.state := state;
	
	// Set the event
	m_pFsmDebugTable^.event := event.event;
	
	// Set the computed time since last state change
	m_pFsmDebugTable^.timeInState := TIME_TO_UDINT(m_StateChangeTimer.GetElapsedTime());
	
	// Reset the state change timer start time
	m_StateChangeTimer.StartNow();
	
END_IF
END_METHOD

END_FUNCTION_BLOCK

// 20 Program Organization Units/Utility Functions/fb_ElapsedTime
(*AUTHOR:			Jaison Schaab*)
(*DATE:				February 26/ 2021*)
(*DESCRIPTION: 		This Function measures the elapsed time from a an indicated start. 
					The elapsed time my be read as LTIME or as TIME by get methods.*)
				
FUNCTION_BLOCK fb_ElapsedTime
VAR_INPUT
END_VAR
VAR_OUTPUT
END_VAR
VAR
	startTime		: ULINT;		// Start time for "F_GetSystemTime()" method
	nsStartTime		: T_DCTIME64;	// Start time for "F_GetCurDcTickTime64()" method
END_VAR

(* ---------------------------------------------------------------------------
Func name   : 	FB_exit
Description : 	Destructor
Inputs      :	None
Returns     : 	None
Notes       : 	
--------------------------------------------------------------------------- *)

METHOD FB_exit
VAR_INPUT
	bInCopyCode : BOOL; // if TRUE, the exit method is called for exiting an instance that is copied afterwards (online change)
END_VAR
// Do nothing
END_METHOD

(* ---------------------------------------------------------------------------
Func name   : 	FB_init
Description : 	Constructor
Inputs      :	None
Returns     : 	None
Notes       : 	
--------------------------------------------------------------------------- *)

METHOD FB_init
VAR_INPUT
	bInitRetains 		: BOOL; 			// if TRUE, the retain variables are initialized (warm start / cold start)
    bInCopyCode  		: BOOL; 			// if TRUE, the instance afterwards gets moved into the copy code (online change)
END_VAR
// Do Nothing
END_METHOD

(* ---------------------------------------------------------------------------
Func name   : 	Disarm
Description : 	Returns the nanoseconds since start of the measurement.
Inputs      :	None
Returns     : 	None
Notes       : 	When more than ~292 years have elapsed, the result would overflow, 
				thus it is clamped to 16#7FFF.FFFF.FFFF.FFFF to indicate the overflow 
				(this is performed for formal reasons rather than for practical ones).
--------------------------------------------------------------------------- *)

METHOD GetElapsedLTime : LTIME
VAR_INPUT
END_VAR
// F_GetSystemTime returns time in 100ns. <JAISON>
GetElapsedLTime := TO_LTIME(MIN(16#7FFFFFFFFFFFFFFF, ((F_GetSystemTime() - startTime) * 100)));		// Convert 100ns to ns by multiplying by 100

// Alternate method, Not Used <JAISON>
// F_GetCurDcTickTime64 returns time in ns. <JAISON>
//GetElapsedLTime	:= TO_LTIME(F_GetCurDcTickTime64() - nsStartTime);								// Result is already in ns
END_METHOD

(* ---------------------------------------------------------------------------
Func name   : 	GetElapsedTime
Description : 	Returns the milliseconds since start of the measurement.
Inputs      :	None
Returns     : 	None
Notes       : 	When more than ~49 days have elapsed, the result would overflow, 
				thus it is clamped to 16#FFFF.FFFF to indicate the overflow.
--------------------------------------------------------------------------- *)

METHOD GetElapsedTime : TIME
VAR_INPUT
END_VAR
VAR CONSTANT
	
END_VAR
// F_GetSystemTime returns time in 100ns. <JAISON>
GetElapsedTime := TO_TIME(MIN(16#FFFFFFFF, ((F_GetSystemTime() - startTime) / 10000)));	// Convert 100ns to ms by multiplying by dividing by 10000

// Alternate method, Not Used <JAISON>
// F_GetCurDcTickTime64 returns time in ns. <JAISON>
//GetElapsedTime	:= TO_TIME((F_GetCurDcTickTime64() - nsStartTime) / 1000000);		// Convert ns to ms by multiplying by dividing by 1000000
END_METHOD

(* ---------------------------------------------------------------------------
Func name   : 	StartNow
Description : 	Sets the start time of the measurement to the actual time.
Inputs      :	None
Returns     : 	None
Notes       : 	
--------------------------------------------------------------------------- *)

METHOD StartNow
VAR_INPUT
END_VAR
// Update the start time variable for both timer methods <JAISON>
startTime	:= F_GetSystemTime();
nsStartTime	:= F_GetCurDcTickTime64();
END_METHOD

END_FUNCTION_BLOCK

// 20 Program Organization Units/Control Functions/PID Functions/PID_StandAlone
(*AUTHOR:		Graham Hunter *)
(*DATE:			Feb 25, 2021 *)
(*DESCRIPTION:	This PID function block is a PID controller with min and max controller output saturation limits WITH PSEUDO anti-integral windup. 
				This integral windup stays CONSTANT over time when staturation occurs so it really gets somewhat UNSTUCK (better than stuck).
				This code has been tested with properly tuned gains on the suction and boost pumps of the E-Frac Ideal Process Plant.*)

(*NOTES:  
INPUTS: 	   					
VAR_IN_OUTs:     				
FUNCTIONALITY: 			  
OUTPUTS:       
EXAMPLE CODE USAGE: 		
*)
(*UPDATE: 				
*)	

FUNCTION_BLOCK PID_StandAlone
VAR_INPUT
	
	rSP				: REAL; // Setpoint
	rFB				: REAL; // Feedback
	rCP				: REAL; // Control Point
	bLimitsActive	: BOOL; // True when CP output limited to min/max, reaches 
	// Here to match HRNU PID format
	rCurrentValue	: REAL;
	rKp				: REAL;
	rKi				: REAL;
	rKd				: REAL;
	
	rMax: REAL; 			// max value of the Control Point (max saturation value)			
	rMin: REAL;				// min value of the Control Point (min saturation value)	
END_VAR
VAR_OUTPUT
	doneInit: BOOL;
END_VAR
VAR
	
	rElapsedTime		: REAL; // [ms], not used currently
	rIntegralWindup		: REAL; // the accumulation of error over time (error*deltaT)
	rError				: REAL;	// Difference between actual feedback value and setpoint
	rPreviousError		: REAL;	// Error from last cycle (for derivitive term)
	rPreviousTime		: LREAL;// [ms]
	lastCycleBelowTarget: BOOL; // Used to clear windup on target pass (not used currently and not coded in properly)
END_VAR

METHOD Execute : REAL
VAR_INPUT
	Feedback		: REAL;	// this is the feedback value
	CurrentValue	: REAL;	// this is the feedforward value (same units as feedback and setpoint values), SET TO 0, DO NOT USE UNLESS YOU KNOW WHAT YOU ARE DOING <GRAHAM>
	Setpoint		: REAL;	// this is the setpoint value
END_VAR
VAR
	// Note: These variables reset after every execute call
	derivative		: REAL;	 // derivative term, delta error divided by delta T
	output			: REAL;	 // this is the PID controller output, whatever units that are required for control of an Actuator [i.e. RPMs to a VFD, Volts to a solenoid valve]
	currentTime		: LREAL; // [ms]
	deltaT			: REAL;  // [s]
END_VAR

// If target surpassed (rising or falling) clear windup, 
// Ken had the right idea but integral windup is when saturation occurs AND the error & output have same sign, this is dead code <GRAHAM>
IF Setpoint > Feedback AND NOT lastCycleBelowTarget THEN//Fall past target
	//rIntegralWindup:=0;
	//UI_Manager.Fell:=TRUE;
	//UI_Manager.Rose:=FALSE;
ELSIF Setpoint < Feedback AND lastCycleBelowTarget THEN//Rise past target
	//rIntegralWindup:=0;
	//UI_Manager.Fell:=FALSE;
	//UI_Manager.Rose:=TRUE;
END_IF

// To accommodate old code format
rSP:=Setpoint;
rFB:=Feedback;
rCurrentValue:=CurrentValue;

currentTime:= TIME_TO_LREAL(TIME());						//ms
deltaT:= LREAL_TO_REAL((currentTime - rPreviousTime)/1000);	//seconds
rError:= rSP - rFB;

IF(NOT doneInit) THEN

	init();
END_IF

//If this hasn't been called in several cycles then reset it
//NOTE: If we ever run slower than 1 Hz this will break PID class
IF deltaT >= 1 THEN
	rIntegralWindup:=0;
	output:=0;
ELSE
	rIntegralWindup:= rIntegralWindup + rError * deltaT;
	derivative:= (rError - rPreviousError) / deltaT;
	
	output:= rCurrentValue + rKp*rError + rKi*rIntegralWindup + rKd*derivative;
	
	IF output > rMax THEN
		// Limit value to max., max saturation occurring
		output:=rMax;
		// reverse latest integral windup, this is somewhat incorrect, the integral windup should be set to zero when saturation occurs AND the error & output have same sign <GRAHAM>
		rIntegralWindup:= rIntegralWindup - rError * deltaT;
		bLimitsActive:= TRUE;
	ELSIF output < rMin THEN
		// Limit value to min, min saturation occurring
		output:=rMin;
		// reverse latest integral windup, this is somewhat incorrect, the integral windup should be set to zero when saturation occurs AND the error & output have same sign <GRAHAM>
		rIntegralWindup:= rIntegralWindup - rError * deltaT;
		bLimitsActive:= TRUE;
	ELSE
		bLimitsActive:= FALSE;
	END_IF
END_IF

//To use for next cycle
rPreviousTime:=currentTime;
rPreviousError:=rError;
//Set control point
rCP:=output;
//return PID output
Execute:=output;

// Used to clear windup on target pass
// this is dead code <GRAHAM>
IF Setpoint > Feedback THEN
	lastCycleBelowTarget:=TRUE;
ELSE
	lastCycleBelowTarget:=FALSE;
END_IF
END_METHOD

METHOD FB_init : BOOL
VAR_INPUT

	bInitRetains	: BOOL;		// if TRUE, the retain variables are initialized (warm start / cold start)
	bInCopyCode		: BOOL;		// if TRUE, the instance afterwards gets moved into the copy code (online change)
END_VAR
	(*
	* Place objects that require initialization here
	* This method is ran once at power up and never again.
	*)
//Default Values

//Input
rKp:= 0;
rKi:= 0;
rKd:= 0;
rMax:= REAL_MAX;
rMin:= -REAL_MAX;

//Output
doneInit:=TRUE;

//Internal
rElapsedTime:=0;
rIntegralWindup:=0;
rError:=0;
rPreviousError:=0;
END_METHOD

METHOD GetGains
VAR_OUTPUT
	Kp: REAL;
	Ki: REAL;
	Kd: REAL;
END_VAR
Kp:=rKp;
Ki:=rKi;
Kd:=rKd;
END_METHOD

METHOD GetLimits
VAR_OUTPUT
	MaxCP: REAL;
	MinCP: REAL;
END_VAR
MaxCP:=rMax;
MinCP:=rMin;
END_METHOD

ACTION init:
rElapsedTime:=0;
rIntegralWindup:=0;
rPreviousError:=0;
doneInit:=true;
END_ACTION

ACTION Reset:
doneInit:=false;
END_ACTION

METHOD SetGains : REAL
VAR_INPUT
	Kp: REAL;
	Ki: REAL;
	Kd: REAL;
END_VAR
rKp:=Kp;
rKi:=Ki;
rKd:=Kd;
END_METHOD

METHOD SetLimits
VAR_INPUT
	MaxCP: REAL;
	MinCP: REAL;
END_VAR
rMax:=MaxCP;
rMin:=MinCP;
END_METHOD

END_FUNCTION_BLOCK

// 20 Program Organization Units/Control Functions/PID Functions/PID_StandAlone_AntiWindup
(*AUTHOR:		Graham Hunter *)
(*DATE:			Feb 25, 2021 *)
(*DESCRIPTION:	This PID function block is a PID controller with min and max controller output saturation limits WITH anti-integral windup. 
				This integral windup is set to zero when staturation occurs and the error AND controller output are the same sign so the controls really get UNSTUCK (better than stuck).
				This code has NOT been tested.*)
				
(*NOTES:  
INPUTS: 	   					
VAR_IN_OUTs:     				
FUNCTIONALITY: 			  
OUTPUTS:       
EXAMPLE CODE USAGE: 		
*)
(*UPDATE: 				
*)	

FUNCTION_BLOCK PID_StandAlone_AntiWindup
VAR_INPUT
	rSP					: REAL; // Setpoint
	rFB					: REAL; // Feedback
	rCP					: REAL; // Control Point
	bLimitsActive		: BOOL; // True when CP output limited to min/max, reaches 
	// Here to match HRNU PID format
	rFeedforwardValue	: REAL;
	rKp					: REAL;
	rKi					: REAL;
	rKd					: REAL;
	
	rMax				: REAL; // max value of the Control Point (max saturation value)			
	rMin				: REAL;	// min value of the Control Point (min saturation value)	
END_VAR
VAR_OUTPUT
	doneInit: BOOL;
END_VAR
VAR
	rElapsedTime		: REAL; // [ms], not used currently
	rIntegralWindup		: REAL; // the accumulation of error over time (error*deltaT)
	rError				: REAL;	// Difference between actual feedback value and setpoint
	rPreviousError		: REAL;	// Error from last cycle (for derivitive term)
	rPreviousTime		: LREAL;// [ms]
	lastCycleBelowTarget: BOOL; // Used to clear windup on target pass (not used currently and not coded in properly)
END_VAR

METHOD Execute : REAL
VAR_INPUT
	Feedback			: REAL;	// this is the feedback value
	FeedforwardValue	: REAL;	// this is the feedforward value (same units as feedback and setpoint values), SET TO 0, DO NOT USE UNLESS YOU KNOW WHAT YOU ARE DOING <GRAHAM>
	Setpoint			: REAL;	// this is the setpoint value
END_VAR
VAR
	// Note: These variables reset after every execute call
	derivative			: REAL;	 // derivative term, delta error divided by delta T
	output				: REAL;	 // this is the PID or controller output, whatever units that are required for control of an Actuator [i.e. RPMs to a VFD, Volts to a solenoid valve]
	currentTime			: LREAL; // [ms]
	deltaT				: REAL;  // [s]
	SignOutputError		: REAL;	 // combination of Output times Error to obtain sign for indication of windup, positive number means error & output have the same sign and integration/windup is increasing 
	
END_VAR
//To accommodate old code format
rSP := Setpoint;
rFB := Feedback;
rFeedforwardValue := FeedforwardValue;

currentTime:= TIME_TO_LREAL(TIME());//ms
deltaT:= LREAL_TO_REAL((currentTime - rPreviousTime)/1000);//seconds
rError:= rSP - rFB;

IF(NOT doneInit) THEN
	init();
END_IF

//If this hasn't been called in several cycles then reset it
//NOTE: If we ever run slower than 1 Hz this will break PID class
IF deltaT >= 1 THEN
	rIntegralWindup:=0;
	output:=0;
ELSE
	rIntegralWindup:= rIntegralWindup + (rError * deltaT);
	derivative:= (rError - rPreviousError) / deltaT;
	
	output := rFeedforwardValue + rKp*rError + rKi*rIntegralWindup + rKd*derivative;
	
	SignOutputError	:= output*rError; // combination of Output times Error to obtain sign to determine if anti-integral windup is required
	
	IF output > rMax THEN
		// Limit value to max., max saturation occurring
		output := rMax;
		bLimitsActive := TRUE;
		
		// Anti-windup, set integral windup to zero when staturation occurs and error AND control output are the same sign (prevent integration/windup from increasing) 
		IF SignOutputError > 0.0 THEN
			rIntegralWindup:= 0.0 - (rError * deltaT);
		END_IF

	ELSIF output < rMin THEN
		// Limit value to min, min saturation occurring
		output:=rMin;
		bLimitsActive:= TRUE;
		
		// Anti-windup, set integral windup to zero when staturation occurs and error AND control output are the same sign (prevent integration/windup from increasing) 
		IF SignOutputError > 0.0 THEN
			rIntegralWindup:= 0.0 - (rError * deltaT);
		END_IF
		
	ELSE
		bLimitsActive:= FALSE;
	END_IF
END_IF

//To use for next cycle
rPreviousTime:=currentTime;
rPreviousError:=rError;

rCP:=output; //Set control point

Execute:=output; //return PID output
END_METHOD

METHOD FB_init : BOOL
VAR_INPUT
	
	bInitRetains	: BOOL; // if TRUE, the retain variables are initialized (warm start / cold start)
	bInCopyCode		: BOOL; // if TRUE, the instance afterwards gets moved into the copy code (online change) 
END_VAR
	(*
	* Place objects that require initialization here
	* This method is ran once at power up and never again.
	*)
//Default Values

//Input
rKp:= 0;
rKi:= 0;
rKd:= 0;
rMax:= REAL_MAX;
rMin:= -REAL_MAX;

//Output
doneInit:=TRUE;

//Internal
rElapsedTime:=0;
rIntegralWindup:=0;
rError:=0;
rPreviousError:=0;
END_METHOD

METHOD GetConfig
VAR_OUTPUT
	Kp: REAL;
	Ki: REAL;
	Kd: REAL;
	MaxCP: REAL;
	MinCP: REAL;
END_VAR
Kp:=rKp;
Ki:=rKi;
Kd:=rKd;

MaxCP:=rMax;
MinCP:=rMin;
END_METHOD

ACTION init:
rElapsedTime:=0;
rIntegralWindup:=0;
rPreviousError:=0;
doneInit:=true;
END_ACTION

ACTION Reset:
doneInit:=false;
END_ACTION

METHOD SetConfig : REAL
VAR_INPUT
	Kp: REAL;
	Ki: REAL;
	Kd: REAL;
	MaxCP: REAL;
	MinCP: REAL;
END_VAR
rKp:=Kp;
rKi:=Ki;
rKd:=Kd;

rMax:=MaxCP;
rMin:=MinCP;
END_METHOD

END_FUNCTION_BLOCK

// 20 Program Organization Units/Control Functions/PID Functions/PID_StandAlone_Stuck
(*AUTHOR:		Graham Hunter *)
(*DATE:			Feb 25, 2021 *)
(*DESCRIPTION:	This PID function block is a PID controller with min and max controller output saturation limits WITHOUT anti-integral windup. 
				This integral windup increases over time when staturation occurs so the controls really gets STUCK at min. or max. controller output saturation limits (not good). 
				This was incorrectly named before as PID_Standalone_Unstuck. This should not be used going forward with new development.
				This code has been tested with properly tuned gains on the Dry Add Augers, Liquid Add Pumps, and Auger Concentration Proppant control of the E-Frac Ideal Process Plant.
*)
				
(*NOTES:  
INPUTS: 	   					
VAR_IN_OUTs:     				
FUNCTIONALITY: 			  
OUTPUTS:       
EXAMPLE CODE USAGE: 		
*)
(*UPDATE: 				
*)	

FUNCTION_BLOCK PID_StandAlone_Stuck
VAR_INPUT
	rSP				: REAL; // Setpoint
	rFB				: REAL; // Feedback
	rCP				: REAL; // Control Point
	bLimitsActive	: BOOL; // True when CP output limited to min/max, reaches 
	// Here to match HRNU PID format
	rCurrentValue	: REAL;
	rKp				: REAL;
	rKi				: REAL;
	rKd				: REAL;
	
	rMax: REAL; 			// max value of the Control Point (max saturation value)			
	rMin: REAL;				// min value of the Control Point (min saturation value)	
END_VAR
VAR_OUTPUT
	doneInit: BOOL;
END_VAR
VAR
	rElapsedTime		: REAL; // [ms], not used currently
	rIntegralWindup		: REAL;	// the accumulation of error over time (error*deltaT)
	rError				: REAL;	// Difference between actual feedback value and setpoint
	rPreviousError		: REAL;	// Error from last cycle (for derivitive term)
	rPreviousTime		: LREAL;// [ms]
	lastCycleBelowTarget: BOOL; // Used to clear windup on target pass (not used currently and not coded in properly)
END_VAR

METHOD Execute : REAL
VAR_INPUT
	Feedback		: REAL;	// this is the feedback value
	CurrentValue	: REAL;	// this is the feedforward value (same units as feedback and setpoint values), SET TO 0, DO NOT USE UNLESS YOU KNOW WHAT YOU ARE DOING <GRAHAM>
	Setpoint		: REAL;	// this is the setpoint value
END_VAR
VAR
	// Note: These variables reset after every execute call
	derivative		: REAL;	 // derivative term, delta error divided by delta T
	output			: REAL;	 // this is the PID or controller output, whatever units that are required for control of an Actuator [i.e. RPMs to a VFD, Volts to a solenoid valve]
	currentTime		: LREAL; // [ms]
	deltaT			: REAL;  // [s]
END_VAR
//To accommodate old code format
rSP:=Setpoint;
rFB:=Feedback;
rCurrentValue:=CurrentValue;

currentTime:= TIME_TO_LREAL(TIME());//ms
deltaT:= LREAL_TO_REAL((currentTime - rPreviousTime)/1000);//seconds
rError:= rSP - rFB;

IF(NOT doneInit) THEN

	init();
END_IF

//If this hasn't been called in several cycles then reset it
//NOTE: If we ever run slower than 1 Hz this will break PID class
IF deltaT >= 1 THEN
	rIntegralWindup:=0;
	output:=0;
ELSE
	rIntegralWindup:= rIntegralWindup + rError * deltaT;
	derivative:= (rError - rPreviousError) / deltaT;
	
	output:= rCurrentValue + rKp*rError + rKi*rIntegralWindup + rKd*derivative;
	
	IF output > rMax THEN
		// Limit value to max., max saturation occurring
		output:=rMax;
		// DON'T reverse latest integral windup, prevents "sticking" at max output, somewhat incorrect, the integral windup should be set to zero when saturation occurs AND the error & output have same sign <GRAHAM>
		// rIntegralWindup:= rIntegralWindup - rError * deltaT;		
		bLimitsActive:= TRUE;
	ELSIF output < rMin THEN
		// Limit value to min, min saturation occurring
		output:=rMin;
		// DON'T reverse latest integral windup, prevents "sticking" at min output, somewhat incorrect, the integral windup should be set to zero when saturation occurs AND the error & output have same sign <GRAHAM>
		//rIntegralWindup:= rIntegralWindup - rError * deltaT;	
		bLimitsActive:= TRUE;
	ELSE
		bLimitsActive:= FALSE;
	END_IF
END_IF

//To use for next cycle
rPreviousTime:=currentTime;
rPreviousError:=rError;

rCP:=output; //Set control point

Execute:=output; //return PID output
END_METHOD

METHOD FB_init : BOOL
VAR_INPUT
	
	bInitRetains	: BOOL; // if TRUE, the retain variables are initialized (warm start / cold start)
	bInCopyCode		: BOOL; // if TRUE, the instance afterwards gets moved into the copy code (online change) 
END_VAR
	(*
	* Place objects that require initialization here
	* This method is ran once at power up and never again.
	*)
//Default Values

//Input
rKp:= 0;
rKi:= 0;
rKd:= 0;
rMax:= REAL_MAX;
rMin:= -REAL_MAX;

//Output
doneInit:=TRUE;

//Internal
rElapsedTime:=0;
rIntegralWindup:=0;
rError:=0;
rPreviousError:=0;
END_METHOD

METHOD GetGains
VAR_OUTPUT
	Kp: REAL;
	Ki: REAL;
	Kd: REAL;
END_VAR
Kp:=rKp;
Ki:=rKi;
Kd:=rKd;
END_METHOD

METHOD GetLimits
VAR_OUTPUT
	MaxCP: REAL;
	MinCP: REAL;
END_VAR
MaxCP:=rMax;
MinCP:=rMin;
END_METHOD

ACTION init:
rElapsedTime:=0;
rIntegralWindup:=0;
rPreviousError:=0;
doneInit:=true;
END_ACTION

ACTION Reset:
doneInit:=false;
END_ACTION

METHOD SetGains : REAL
VAR_INPUT
	Kp: REAL;
	Ki: REAL;
	Kd: REAL;
END_VAR
rKp:=Kp;
rKi:=Ki;
rKd:=Kd;
END_METHOD

METHOD SetLimits
VAR_INPUT
	MaxCP: REAL;
	MinCP: REAL;
END_VAR
rMax:=MaxCP;
rMin:=MinCP;
END_METHOD

END_FUNCTION_BLOCK

// 20 Program Organization Units/Equipment Functions/TriStateValve/fb_AnalogFeedbackValve
(*AUTHOR:			Jaison Schaab*)
(*DATE:				March. 12 / 2020*)
(*DESCRIPTION: 		This function block provides the functionality for a Tri-State valve which
					has analog valve position feedback.  This valve is controlled by output
					boolean Open/Close actuators.  The user will supply configurable values for
					valve Open/Close which will be used to determine the valves state.*)
				
(*NOTES:			The Open value can be smaller, larger or equal to the Close value.
					The logic will automatically decode the valve state in any scaling
					situaltion.
*)

(*UPDATE: 			March. 23 2021 - Jaison Schaab

					Code Is fully tested and functional.				
*)

(*UPDATE: 			March. 18 2021 - Jaison Schaab

					Code Ported from Wago.
					
					Code has NOT Yet been tested.
*)

(*UPDATE: 			September. 3 2020 - Jaison Schaab

					Added a "IsShifting" method for use in the control class development to detect when valve is shifting.
*)

(*UPDATE: 			September. 1 2020 - Jaison Schaab

					Added a "IsShiftingError" method for use in the control class development to detect valve shift error.
*)

(*UPDATE: 			April. 28 2020 - Jaison Schaab

					Added the InitAlarms function which now NEEDS to be called in order to properly hook up the alarm monitors.
					This method is required because codesys does NOT properly propogate the FB_Init information like constructors
					in C code, so it is impossible to pass down the devceId information.
*)

FUNCTION_BLOCK fb_AnalogFeedbackValve
VAR_INPUT
	xEnable						: BOOL;						// Enable inputs and valve operation
	OpenCommand					: BOOL;						// Open valve command input
	CloseCommand				: BOOL;						// Close valve command input
	InitialValvePosition		: TValveTriStatePosition;	// Position the valve will shift to when enabled (To be retianed if desired outside this block)
	ValveFeedback				: REAL;
	OpenLimit					: REAL;
	CloseLimit					: REAL;
	ValveShiftTimeout			: TIME;						// Valve shift timout value
END_VAR
VAR_OUTPUT
	ValvePosition				: TValveTriStatePosition;	// Current valve position	(0 = closed, 1 = open)
	OpenActuator				: BOOL;						// Valve open actuator (TRUE to OPEN valve)
	CloseActuator				: BOOL;						// Valve close actuator (TRUE to CLOSE valve)
END_VAR
VAR
	(* TriState Valve Function Block *)	

	m_TriStateValve				: fb_TriStateValve;			// Tri-State valve common control with state machine
	
	(* Valve Status *)	
	m_OpenedFeedback			: BOOL;						// Internal valve opened feedback
	m_ClosedFeedback			: BOOL;						// Internal valve closed feedback
	
	OpenBiStable				: RS;						// Triggers for valve opened feedback logic
	CloseBiStable				: RS;						// Triggers for valve closed feedback logic
	
	m_ValveShiftError			: BOOL;						// Valve shift timeout error flag
	
	(* Alarms *)
	m_ValveShiftTimeout			: fb_AlarmMonitor;			// Alarm monitor for valve shift timeout error
	
	(* Event Triggers *)	

	m_EnableTrigger				: R_TRIG;					// Valve enabled trigger
	m_DisableTrigger			: F_TRIG;					// Valve disabled trigger
	m_OpenTrigger				: R_TRIG;					// Valve open trigger
	m_CloseTrigger				: R_TRIG;					// Valve close trigger

END_VAR

// Run the common TriState Valve function block which manages the state machine
m_TriStateValve(	xEnable					:= xEnable,
					InitialValvePosition	:= InitialValvePosition,
					Opened_Feedback			:= m_OpenedFeedback, 
					Closed_Feedback			:= m_ClosedFeedback, 
					ValveShiftTimeout		:= ValveShiftTimeout,
					ValvePosition			=> ValvePosition, 
					Open_Actuator			=> OpenActuator, 
					Close_Actuator			=> CloseActuator, 
					ShiftingError			=> m_ValveShiftError);
					
// (* EVENT TRIGGERS *)

// Valve enabled trigger
m_EnableTrigger(CLK:= xEnable);
IF (m_EnableTrigger.Q)THEN

	// Disable the actuator outputs
	OpenActuator := FALSE;	
	CloseActuator := FALSE;

	// Clear all event triggers to ensure all events are captured on startup
	// NOTE: DO NOT RESET ENABLE/DISABLE TRIGGERS <JAISON>
	m_OpenTrigger(CLK:= FALSE);
	m_CloseTrigger(CLK:= FALSE);
	
END_IF

// Valve disabled trigger
m_DisableTrigger(CLK:= xEnable);
IF (m_DisableTrigger.Q)THEN
	// Disable the alarm monitor
	m_ValveShiftTimeout.DisableLimit();
END_IF

// Open valve command event trigger <JAISON>
m_OpenTrigger(CLK:= OpenCommand);
IF (m_OpenTrigger.Q) THEN
	OpenValve();
END_IF

// Close valve command event trigger <JAISON>
m_CloseTrigger(CLK:= CloseCommand);
IF (m_CloseTrigger.Q) THEN
	CloseValve();
END_IF

// (* VALVE FEEDBACK *)

// Decode the valve feedback <JAISON>
IF ((CloseLimit > OpenLimit) AND xEnable) THEN // CLOSE > OPEN CASE
	
	OpenBiStable(SET:= (ValveFeedback <= OpenLimit), RESET1:= (ValveFeedback > OpenLimit), Q1=> m_OpenedFeedback);
	CloseBiStable(SET:= (ValveFeedback >= CloseLimit), RESET1:= (ValveFeedback < CloseLimit), Q1=> m_ClosedFeedback);

ELSIF ((CloseLimit < OpenLimit) AND xEnable) THEN // CLOSE < OPEN CASE

	OpenBiStable(SET:= (ValveFeedback >= OpenLimit), RESET1:= (ValveFeedback < OpenLimit), Q1=> m_OpenedFeedback);
	CloseBiStable(SET:= (ValveFeedback <= CloseLimit), RESET1:= (ValveFeedback > CloseLimit), Q1=> m_ClosedFeedback);

ELSE // CLOSE = OPEM CASE
	
	OpenBiStable(SET:= (ValveFeedback > OpenLimit), RESET1:= (ValveFeedback < OpenLimit), Q1=> m_OpenedFeedback);
	CloseBiStable(SET:= (ValveFeedback < CloseLimit), RESET1:= (ValveFeedback > CloseLimit), Q1=> m_ClosedFeedback);

END_IF

// Run the Alarm Monitors <JAISON>
m_ValveShiftTimeout.MonitorBool(value:= m_ValveShiftError);

(* ---------------------------------------------------------------------------
Func name   : 	CloseValve
Description : 	Sends an valve close event the the Tri-State 
				valve if the block is Enabled.
Inputs      :	None
Returns     : 	None
Notes       : 	This method should be triggered by an event 
				and not called cyclically to prevent flooding 
				the FSM event Queue.
--------------------------------------------------------------------------- *)

METHOD CloseValve : BOOL
VAR_INPUT
END_VAR
// Send CLOSE command to Tri-State Valve FSM if the valve is enabled
IF xEnable THEN
	m_TriStateValve.CloseValve();
END_IF
END_METHOD

(* ---------------------------------------------------------------------------
Func name   : 	FB_exit
Description : 	Destructor
Inputs      :	None
Returns     : 	None
Notes       : 	
--------------------------------------------------------------------------- *)

METHOD FB_exit : BOOL
VAR_INPUT
	bInCopyCode : BOOL; // if TRUE, the exit method is called for exiting an instance that is copied afterwards (online change)
END_VAR
// Do Nothing
END_METHOD

(* ---------------------------------------------------------------------------
Func name   : 	FB_init
Description : 	Constructor
Inputs      :	None
Returns     : 	None
Notes       : 	
--------------------------------------------------------------------------- *)

METHOD FB_init : BOOL
VAR_INPUT
	bInitRetains 		: BOOL; 				// if TRUE, the retain variables are initialized (warm start / cold start)
    bInCopyCode  		: BOOL; 				// if TRUE, the instance afterwards gets moved into the copy code (online change)
END_VAR
// Disable the actuator outputs
OpenActuator := FALSE;	
CloseActuator := FALSE;

// Clear all event triggers to ensure all events are captured on startup
m_EnableTrigger(CLK:= FALSE);
m_DisableTrigger(CLK:= FALSE);
m_OpenTrigger(CLK:= FALSE);
m_CloseTrigger(CLK:= FALSE);
END_METHOD

(* ---------------------------------------------------------------------------
Func name   : 	InitAlarms
Description : 	Initializes the alarm monitors for the valve.
Inputs      :	devId	:	Device Id used for alarm integration
Returns     : 	None
Notes       : 	
--------------------------------------------------------------------------- *)

METHOD InitAlarms
VAR_INPUT
	devId	: UDeviceId;	// Device Id used for alarm integration
END_VAR
// Initialize the alarm monitors and set their limits
m_ValveShiftTimeout.InitAlarm(code:= f_AlarmCode(devId, f_FaultCode(TFaultPriority.Warning, TFaultCondition.TimeOut)), alarmType:= TAlarmMonitorType.upper_limit, delayTime:= T#1S);
m_ValveShiftTimeout.SetLimitBool(on:= TRUE, off:= FALSE);
m_ValveShiftTimeout.EnableLimit();
END_METHOD

(* ---------------------------------------------------------------------------
Func name   : 	IsClosed
Description : 	Polls valve for its closed status.
Inputs      :	None
Returns     : 	BOOL	-	TRUE is valve Closed, FALSE otherwise
Notes       : 	
--------------------------------------------------------------------------- *)

METHOD IsClosed : BOOL
VAR_INPUT
END_VAR
IsClosed := m_ClosedFeedback;
END_METHOD

(* ---------------------------------------------------------------------------
Func name   : 	IsOpened
Description : 	Polls valve for its opened status.
Inputs      :	None
Returns     : 	BOOL	-	TRUE is valve Opened, FALSE otherwise
Notes       : 	
--------------------------------------------------------------------------- *)

METHOD IsOpened : BOOL
VAR_INPUT
END_VAR
IsOpened := m_OpenedFeedback;
END_METHOD

(* ---------------------------------------------------------------------------
Func name   : 	IsShifting
Description : 	Polls valve for its shifting status.
Inputs      :	None
Returns     : 	BOOL	-	TRUE is valve is shifting, FALSE otherwise
Notes       : 	
--------------------------------------------------------------------------- *)

METHOD IsShifting : BOOL
VAR_INPUT
END_VAR
IF (ValvePosition = TValveTriStatePosition.PosUnknown) THEN
	IsShifting := TRUE;
ELSE
	IsShifting := FALSE;
END_IF
END_METHOD

(* ---------------------------------------------------------------------------
Func name   : 	IsShiftingError
Description : 	Polls valve for its shifting error status.
Inputs      :	None
Returns     : 	BOOL	-	TRUE is valve shift error, FALSE otherwise
Notes       : 	
--------------------------------------------------------------------------- *)

METHOD IsShiftingError : BOOL
VAR_INPUT
END_VAR
IsShiftingError	:= m_ValveShiftError;
END_METHOD

(* ---------------------------------------------------------------------------
Func name   : 	OpenValve
Description : 	Sends an valve open event the the Tri-State
				valve if the block is Enabled.
Inputs      :	None
Returns     : 	None
Notes       : 	This method should be triggered by an event 
				and not called cyclically to prevent flooding 
				the FSM event Queue.
--------------------------------------------------------------------------- *)

METHOD OpenValve : BOOL
VAR_INPUT
END_VAR
// Send OPEN command to Tri-State Valve FSM if the valve is enabled
IF xEnable THEN
	m_TriStateValve.OpenValve();
END_IF
END_METHOD

END_FUNCTION_BLOCK

// 20 Program Organization Units/Equipment Functions/TriStateValve/fb_TriStateValve
(*AUTHOR:			Jaison Schaab*)
(*DATE:				March. 9 / 2020*)
(*DESCRIPTION: 		This function block provides the base functionality for a Tri-State valve, which
					wassumes boolean feedback for Open/Close.  This valve utilizes a table driven FSM
					to capture the events and control the output boolean Open/Close actuators. *)

(*UPDATE: 			March. 23 2021 - Jaison Schaab

					Code Is fully tested and functional.				
*)

(*UPDATE: 			March. 18 2021 - Jaison Schaab

					Code Ported from Wago.
					
					Code has NOT Yet been tested.
*)

(*UPDATE: 			July. 31 2020 - Jaison Schaab

					Fixed an issue discovered by Ryan during the development of the dual action valve.
					
					The valve shifting timeout value was previously ONLY reset once the valve successfully
					shifted; this meant that if the valve was stuck and subsequent open/close commands
					were issued, the timeout would not reset and the outputs would remain on.  

					To fix this the valve shift timeout now resets when an open/close command is issued 
					and the timerwill start again.
*)	
				
FUNCTION_BLOCK fb_TriStateValve IMPLEMENTS i_actionHandler
VAR_INPUT
	xEnable						: BOOL;						// Enable inputs and FSM operation
	InitialValvePosition		: TValveTriStatePosition;	// Position the valve will shift to when enabled (To be retianed if desired outside this block)
	Opened_Feedback				: BOOL;						// Valve opened feedback input
	Closed_Feedback				: BOOL;						// Valve closed feedback input
	ValveShiftTimeout			: TIME;						// Valve shift timout value input
END_VAR
VAR_OUTPUT
	ValvePosition				: TValveTriStatePosition;	// Current valve position	(0 = closed, 1 = open)
	Open_Actuator				: BOOL;						// Valve open actuator			
	Close_Actuator				: BOOL;						// Valve close actuator
	ShiftingError				: BOOL;						// Shifting error bit (TRUE when shifting timeout expired) Can be used for alarm
	FsmError					: BOOL;						// Fsm Error (TRUE when FSM errors) Can be used for alarm, FSM will be auto-reset 
END_VAR
VAR

	(* Event Triggers *)	

	m_EnableTrigger				: R_TRIG;					// Valve enabled event trigger
	m_DisableTrigger			: F_TRIG;					// Valve disabled event trigger
	m_OpenedTrigger				: R_TRIG;					// Valve opened event trigger
	m_ClosedTrigger				: R_TRIG;					// Valve closed event trigger
	m_PositionMismatchTrigger	: R_TRIG;					// Valve position mismatch event trigger
	m_ShiftTimeoutTrigger		: R_TRIG;					// Valve shift timeout event trigger
	
	m_ShiftTimer				: TON;						// Valve shift timer used to detect timeout error
	
	(* Valve Status *)
	m_ValveCmdPosition			: TValveTriStatePosition;	// Valve last commanded position
		
	(* Finite State Machine *)
													
	m_TriStateValveFsmTable		: ARRAY [0..FSM_STATE_ARRAY_MAX, 0..FSM_EVENT_ARRAY_MAX, 0..FSM_ACTIONS_ARRAY_MAX] OF BYTE := [
	
	(* FsmState_Error ------------------------------------------------------------------------- *)
	(*  Next State											Action		                        *)
	
		(* FsmEvent_ValveEnable *)
		FSM_EVENT_INVALID,									TriStateValveFsmAction.FsmAction_None,
                          
		(* FsmEvent_ValveDisable *)
		FSM_EVENT_INVALID,									TriStateValveFsmAction.FsmAction_None,
	
		(* FsmEvent_ValveOpen *)
		FSM_EVENT_INVALID,									TriStateValveFsmAction.FsmAction_None,

		(* FsmEvent_ValveClose *)  
		FSM_EVENT_INVALID,									TriStateValveFsmAction.FsmAction_None,
			
		(* FsmEvent_ValveOpened *)
		FSM_EVENT_INVALID,									TriStateValveFsmAction.FsmAction_None,

		(* FsmEvent_ValveClosed *)
		FSM_EVENT_INVALID,									TriStateValveFsmAction.FsmAction_None,

		(* FsmEvent_ValveShiftTimerExpired *)
		FSM_EVENT_INVALID,									TriStateValveFsmAction.FsmAction_None,
		
		(* FsmEvent_ValvePositionMismatch *)
		FSM_EVENT_INVALID,									TriStateValveFsmAction.FsmAction_None
	,
	
	(* FsmState_ValveOff ---------------------------------------------------------------------- *)
	(*  Next State											Action		                        *)
	
		(* FsmEvent_ValveEnable *)
		TriStateValveFsmState.FsmState_ValveShifting,		TriStateValveFsmAction.FsmAction_ValveEnabled,
                          
		(* FsmEvent_ValveDisable *)
		TriStateValveFsmState.FsmState_ValveOff,			TriStateValveFsmAction.FsmAction_None,
	
		(* FsmEvent_ValveOpen *)
		TriStateValveFsmState.FsmState_ValveOff,			TriStateValveFsmAction.FsmAction_None,
                          
		(* FsmEvent_ValveClose *)
		TriStateValveFsmState.FsmState_ValveOff,			TriStateValveFsmAction.FsmAction_None,
		
		(* FsmEvent_ValveOpened *)
		TriStateValveFsmState.FsmState_ValveOff,			TriStateValveFsmAction.FsmAction_None,
                          
		(* FsmEvent_ValveClosed *)
		TriStateValveFsmState.FsmState_ValveOff,			TriStateValveFsmAction.FsmAction_None,
                          
		(* FsmEvent_ValveShiftTimerExpired *)
		TriStateValveFsmState.FsmState_ValveOff,			TriStateValveFsmAction.FsmAction_None,
		
		(* FsmEvent_ValvePositionMismatch *)
		TriStateValveFsmState.FsmState_ValveOff,			TriStateValveFsmAction.FsmAction_None
  	,

	(* FsmState_ValveClosed ------------------------------------------------------------------- *)
	(*  Next State											Action		                        *)
	
		(* FsmEvent_ValveEnable *)
		TriStateValveFsmState.FsmState_ValveClosed,			TriStateValveFsmAction.FsmAction_None,
                          
		(* FsmEvent_ValveDisable *)
		TriStateValveFsmState.FsmState_ValveOff,			TriStateValveFsmAction.FsmAction_ValveDisabled,
	
		(* FsmEvent_ValveOpen *)
		TriStateValveFsmState.FsmState_ValveShifting,		TriStateValveFsmAction.FsmAction_ValveOpen,
                          
		(* FsmEvent_ValveClose *)
		TriStateValveFsmState.FsmState_ValveClosed,			TriStateValveFsmAction.FsmAction_None,
		
		(* FsmEvent_ValveOpened *)
		FSM_EVENT_INVALID,									FSM_ACTION_UNEXPECTED_EVENT,
                          
		(* FsmEvent_ValveClosed *)
		TriStateValveFsmState.FsmState_ValveClosed,			TriStateValveFsmAction.FsmAction_None,
                          
		(* FsmEvent_ValveShiftTimerExpired *)
		FSM_EVENT_INVALID,									FSM_ACTION_UNEXPECTED_EVENT,
		
		(* FsmEvent_ValvePositionMismatch *)
		TriStateValveFsmState.FsmState_ValveShifting,		TriStateValveFsmAction.FsmAction_ValvePositionMismatch
  	,

	(* FsmState_ValveOpened ------------------------------------------------------------------- *)
	(*  Next State											Action		                        *)
	
		(* FsmEvent_ValveEnable *)
		TriStateValveFsmState.FsmState_ValveOpened,			TriStateValveFsmAction.FsmAction_None,
                          
		(* FsmEvent_ValveDisable *)
		TriStateValveFsmState.FsmState_ValveOff,			TriStateValveFsmAction.FsmAction_ValveDisabled,
	
		(* FsmEvent_ValveOpen *)
		TriStateValveFsmState.FsmState_ValveOpened,			TriStateValveFsmAction.FsmAction_None,
                           
		(* FsmEvent_ValveClose *)
		TriStateValveFsmState.FsmState_ValveShifting,		TriStateValveFsmAction.FsmAction_ValveClose,
		
		(* FsmEvent_ValveOpened *)
		TriStateValveFsmState.FsmState_ValveOpened,			TriStateValveFsmAction.FsmAction_None,
                           
		(* FsmEvent_ValveClosed *)
		FSM_EVENT_INVALID,									FSM_ACTION_UNEXPECTED_EVENT,
                           
		(* FsmEvent_ValveShiftTimerExpired *)
		FSM_EVENT_INVALID,									FSM_ACTION_UNEXPECTED_EVENT,
		
		(* FsmEvent_ValvePositionMismatch *)
		TriStateValveFsmState.FsmState_ValveShifting,		TriStateValveFsmAction.FsmAction_ValvePositionMismatch
	,

	(* FsmState_ValveShifting ----------------------------------------------------------------- *)
	(*  Next State											Action		                        *)
	
		(* FsmEvent_ValveEnable *)
		TriStateValveFsmState.FsmState_ValveShifting,		TriStateValveFsmAction.FsmAction_None,
                          
		(* FsmEvent_ValveDisable *)
		TriStateValveFsmState.FsmState_ValveOff,			TriStateValveFsmAction.FsmAction_ValveDisabled,
	
		(* FsmEvent_ValveOpen *)
		TriStateValveFsmState.FsmState_ValveShifting,		TriStateValveFsmAction.FsmAction_ValveOpen,
                      
		(* FsmEvent_ValveClose *) 
		TriStateValveFsmState.FsmState_ValveShifting,		TriStateValveFsmAction.FsmAction_ValveClose,
		
		(* FsmEvent_ValveOpened *)
		TriStateValveFsmState.FsmState_ValveOpened,			TriStateValveFsmAction.FsmAction_ValveOpened,
                      
		(* FsmEvent_ValveClosed *)
		TriStateValveFsmState.FsmState_ValveClosed,			TriStateValveFsmAction.FsmAction_ValveClosed,
                      
		(* FsmEvent_ValveShiftTimerExpired *)
		TriStateValveFsmState.FsmState_ValveShifting,		TriStateValveFsmAction.FsmAction_ValveShiftTimerExpired,
		
		(* FsmEvent_ValvePositionMismatch *)
		TriStateValveFsmState.FsmState_ValveShifting,		TriStateValveFsmAction.FsmAction_ValvePositionMismatch
  
	];
	
	m_TriStateValveControlFSM	: fb_FSM(	fsmId			:= ADR(m_TriStateValveControlFSM),
											stateTable		:= ADR(m_TriStateValveFsmTable),
											actionHandler	:= THIS^, 	// Use a self pointer in order to keep the action handler routine (ExecuteAction) in same function block <JAISON>
											numStates		:= TriStateValveFsmState.NUM_FsmTriStateValveStates,
											numEvents		:= TriStateValveFsmEvent.NUM_FsmTriStateValveEvents,
											initialState	:= TriStateValveFsmState.FsmState_ValveOff);
											
	m_FsmError					: BOOL;						// FSM error bit (TRUE = FSM Halted)
	m_FsmErrorNum				: TFsmError;				// FSM error ENUM number
	m_FsmCurrentState			: TriStateValveFsmState;	// Current FSM state output
	m_FsmLastState				: TriStateValveFsmState;	// Previous state used for debugging FSM errors
	m_FsmLastEvent				: TriStateValveFsmEvent;	// Last triggered event output
	m_FsmLastAction				: TriStateValveFsmAction;	// Last run action output

END_VAR
VAR CONSTANT
	
	(* Finite State Machine *)

	(* ----------------------------------------------------------------------------
	Const name  : FSM_NUM_EVENT_ACTIONS
	Description : Maximum number of actions that are to be executed for each event 
				  Must be at least 1 action defined				
	Notes       : Used in FSM table definitions
	---------------------------------------------------------------------------- *)
	FSM_NUM_EVENT_ACTIONS: INT := 1;
	
	(* ----------------------------------------------------------------------------
	Const name  : FSM_NUM_STATES
	Description : Total number of states 
	Notes       : Used in FSM table definitions
	---------------------------------------------------------------------------- *)
	FSM_NUM_STATES: INT := TriStateValveFsmState.NUM_FsmTriStateValveStates;
	
	(* ----------------------------------------------------------------------------
	Const name  : FSM_NUM_EVENTS
	Description : Total number of events per state
	Notes       : Used in FSM table definitions
	---------------------------------------------------------------------------- *)
	FSM_NUM_EVENTS: INT := TriStateValveFsmEvent.NUM_FsmTriStateValveEvents;
	
	(* ----------------------------------------------------------------------------
	Const name  : FSM_STATE_ARRAY_MAX
	Description : Max state array index value in the FSM table
				  Must subtract 1 due to arrays starting at 0
	Notes       : Used in FSM table definitions
	---------------------------------------------------------------------------- *)
	FSM_STATE_ARRAY_MAX: INT := FSM_NUM_STATES - 1;
	
